KUKA KRL program: EPS_2_25369_MH1A_A_20251128065454.src

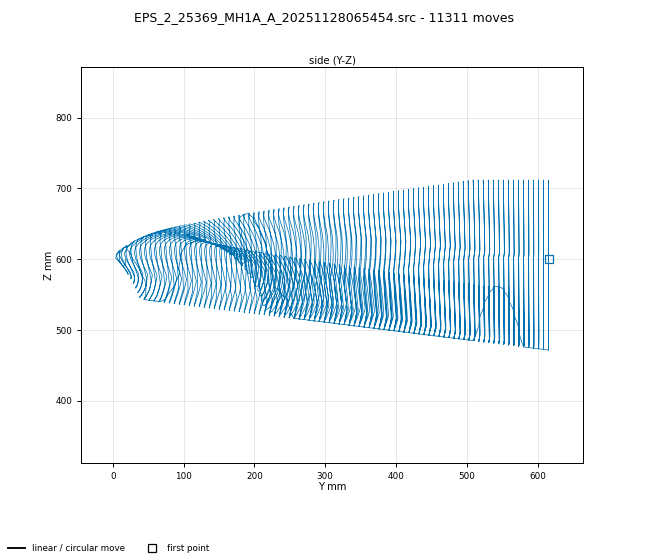
[picture p0: tool path of EPS_2_25369_MH1A_A_20251128065454.src, 11311 of 11313 moves have a stored position in this frame; points joined in program order, loops and branches not executed]
&ACCESS RVP
&REL 4
&COMMENT QRS 19112012
&PARAM EDITMASK = *
DEF PART()
EXT BAS (BAS_COMMAND :IN,REAL :IN )
INT I
BAS (#INITMOV,0 )

;KUKA QRS Post kuka4.cps  Date:22-06-2017 !

File_ID=2931

QRS_PRE_INIT()

;Init var - Until changes are made in qrs_pre_init
Outlet_Square_prg=0
Inlet_1_Square_prg=0
Inlet_2_Square_prg=0
Inlet_3_Square_prg=0
Inlet_4_Square_prg=0
Inlet_5_Square_prg=0

Outlet_1={X 0.000, Y 509.750, Z 611.500, B 0.000, E1 0.000 }
Inlet_1={X 0.000, Y 524.260, Z 411.500, B 0.000, E1 124.000 }
Outlet_1_type=201
Inlet_1_type=201
;QRS#1=Sidecore dimensions
;QRS#2=200-8" PVC SDR 35
;QRS#3=200-8" PVC SDR 35
;QRS#4=
;QRS#5=
;QRS#6=
;QRS#7=
;QRS#8=
;QRS#9=12-08 PSX
;QRS#10=12-08 PSX
;QRS#11=
;QRS#12=
;QRS#13=
;QRS#14=
;QRS#15=
;QRS#16=1220x127x991 3,25'
;QRS#17=EPS Height
;QRS#18=712
;QRS#19=*
;QRS#20= UPDATED VERSION 22-06-2017
;QRS#21=*
Outlet_Square=0100
Inlet_1_Square=0100
Inlet_2_Square=0
Inlet_3_Square=0
Inlet_4_Square=0
Inlet_5_Square=0
Mill_Square=1
Outlet_Square_Prg=204
Inlet_1_Square_prg=204

QRS_INIT()

$ADVANCE=5

; T1
PTP {E1 173.629,E2 173.629}
PTP {X 0,Y 615.476,A -85,B 0,C 180,E1 173.629,E2 173.629,E3 0,E4 0,E5 0,E6 0}
QRS_SPEED_INIT()
LIN {X 0,Y 615.476,Z 600,A -85,B 0,C 180,E1 173.629,E2 173.629,E3 0,E4 0,E5 0,E6 0} C_VEL
LIN {X 0,Y 615.476,Z 481.876,A -85,B 0,C 180,E1 173.629,E2 173.629} C_VEL
LIN {X 0,Y 615.476,Z 473.699,A -85,B 0,C 180,E1 173.629,E2 173.629} C_VEL
LIN {X 0,Y 615.467,Z 471.699,A -85,B 0,C 180,E1 173.442,E2 173.442} C_VEL
LIN {X 0,Y 615.466,Z 471.7,A -85,B 0,C 180,E1 170.801,E2 170.801} C_VEL
LIN {X 0,Y 615.488,Z 471.697,A -85,B 0,C 180,E1 168.139,E2 168.139} C_VEL
LIN {X 0,Y 615.489,Z 471.7,A -85,B 0,C 180,E1 165.451,E2 165.451} C_VEL
LIN {X 0,Y 615.49,Z 471.699,A -85,B 0,C 180,E1 162.729,E2 162.729} C_VEL
LIN {X 0,Y 615.492,Z 471.695,A -85,B 0,C 180,E1 159.967,E2 159.967} C_VEL
LIN {X 0,Y 615.461,Z 471.832,A -85,B 0,C 180,E1 157.233,E2 157.233} C_VEL
LIN {X 0,Y 615.482,Z 484.752,A -85,B 0,C 180,E1 156.799,E2 156.799} C_VEL
LIN {X 0,Y 615.487,Z 496.263,A -85,B 0,C 180,E1 156.274,E2 156.274} C_VEL
LIN {X 0,Y 615.488,Z 507.199,A -85,B 0,C 180,E1 155.638,E2 155.638} C_VEL
LIN {X 0,Y 615.498,Z 517.865,A -85,B 0,C 180,E1 154.864,E2 154.864} C_VEL
LIN {X 0,Y 615.497,Z 526.422,A -85,B 0,C 180,E1 154.103,E2 154.103} C_VEL
LIN {X 0,Y 615.499,Z 535.499,A -85,B 0,C 180,E1 153.105,E2 153.105} C_VEL
LIN {X 0,Y 615.497,Z 542.974,A -85,B 0,C 180,E1 152.085,E2 152.085} C_VEL
LIN {X 0,Y 615.497,Z 549.38,A -85,B 0,C 180,E1 150.969,E2 150.969} C_VEL
LIN {X 0,Y 615.495,Z 554.304,A -85,B 0,C 180,E1 149.84,E2 149.84} C_VEL
LIN {X 0,Y 615.493,Z 557.321,A -85,B 0,C 180,E1 148.914,E2 148.914} C_VEL
LIN {X 0,Y 615.496,Z 560.023,A -85,B 0,C 180,E1 147.669,E2 147.669} C_VEL
LIN {X 0,Y 615.494,Z 561.269,A -85,B 0,C 180,E1 146.466,E2 146.466} C_VEL
LIN {X 0,Y 615.497,Z 561.091,A -85,B 0,C 180,E1 145.185,E2 145.185} C_VEL
LIN {X 0,Y 615.496,Z 559.897,A -85,B 0,C 180,E1 144.166,E2 144.166} C_VEL
LIN {X 0,Y 615.495,Z 557.5,A -85,B 0,C 180,E1 143.063,E2 143.063} C_VEL
LIN {X 0,Y 615.497,Z 553.786,A -85,B 0,C 180,E1 141.932,E2 141.932} C_VEL
LIN {X 0,Y 615.497,Z 549.361,A -85,B 0,C 180,E1 140.937,E2 140.937} C_VEL
LIN {X 0,Y 615.497,Z 543.531,A -85,B 0,C 180,E1 139.91,E2 139.91} C_VEL
LIN {X 0,Y 615.495,Z 536.324,A -85,B 0,C 180,E1 138.905,E2 138.905} C_VEL
LIN {X 0,Y 615.498,Z 527.522,A -85,B 0,C 180,E1 137.919,E2 137.919} C_VEL
LIN {X 0,Y 615.499,Z 517.785,A -85,B 0,C 180,E1 137.04,E2 137.04} C_VEL
LIN {X 0,Y 615.492,Z 507.415,A -85,B 0,C 180,E1 136.286,E2 136.286} C_VEL
LIN {X 0,Y 615.48,Z 496.612,A -85,B 0,C 180,E1 135.654,E2 135.654} C_VEL
LIN {X 0,Y 615.493,Z 484.907,A -85,B 0,C 180,E1 135.117,E2 135.117} C_VEL
LIN {X 0,Y 615.477,Z 471.697,A -85,B 0,C 180,E1 134.663,E2 134.663} C_VEL
LIN {X 0,Y 615.488,Z 471.701,A -85,B 0,C 180,E1 132.08,E2 132.08} C_VEL
LIN {X 0,Y 615.483,Z 471.692,A -85,B 0,C 180,E1 129.751,E2 129.751} C_VEL
LIN {X 0,Y 615.466,Z 471.7,A -85,B 0,C 180,E1 127.244,E2 127.244} C_VEL
LIN {X 0,Y 615.483,Z 471.7,A -85,B 0,C 180,E1 124.699,E2 124.699} C_VEL
LIN {X 0,Y 615.476,Z 471.694,A -85,B 0,C 180,E1 122.328,E2 122.328} C_VEL
LIN {X 0,Y 615.454,Z 471.699,A -85,B 0,C 180,E1 119.408,E2 119.408} C_VEL
LIN {X 0,Y 615.497,Z 471.7,A -85,B 0,C 180,E1 117.046,E2 117.046} C_VEL
LIN {X 0,Y 615.474,Z 471.701,A -85,B 0,C 180,E1 114.273,E2 114.273} C_VEL
LIN {X 0,Y 615.482,Z 471.696,A -85,B 0,C 180,E1 111.432,E2 111.432} C_VEL
LIN {X 0,Y 615.47,Z 471.7,A -85,B 0,C 180,E1 109.339,E2 109.339} C_VEL
LIN {X 0,Y 615.491,Z 471.702,A -85,B 0,C 180,E1 106.587,E2 106.587} C_VEL
LIN {X 0,Y 615.495,Z 471.695,A -85,B 0,C 180,E1 103.874,E2 103.874} C_VEL
LIN {X 0,Y 615.474,Z 471.699,A -85,B 0,C 180,E1 100.878,E2 100.878} C_VEL
LIN {X 0,Y 615.47,Z 471.695,A -85,B 0,C 180,E1 98.537,E2 98.537} C_VEL
LIN {X 0,Y 615.487,Z 471.697,A -85,B 0,C 180,E1 95.899,E2 95.899} C_VEL
LIN {X 0,Y 615.491,Z 471.698,A -85,B 0,C 180,E1 93.273,E2 93.273} C_VEL
LIN {X 0,Y 615.452,Z 471.7,A -85,B 0,C 180,E1 90.654,E2 90.654} C_VEL
LIN {X 0,Y 615.498,Z 471.689,A -85,B 0,C 180,E1 88.037,E2 88.037} C_VEL
LIN {X 0,Y 615.471,Z 471.7,A -85,B 0,C 180,E1 85.415,E2 85.415} C_VEL
LIN {X 0,Y 615.482,Z 471.701,A -85,B 0,C 180,E1 82.784,E2 82.784} C_VEL
LIN {X 0,Y 615.486,Z 471.693,A -85,B 0,C 180,E1 80.138,E2 80.138} C_VEL
LIN {X 0,Y 615.461,Z 471.697,A -85,B 0,C 180,E1 77.469,E2 77.469} C_VEL
LIN {X 0,Y 615.487,Z 471.696,A -85,B 0,C 180,E1 75.451,E2 75.451} C_VEL
LIN {X 0,Y 615.453,Z 471.7,A -85,B 0,C 180,E1 72.728,E2 72.728} C_VEL
LIN {X 0,Y 615.491,Z 471.69,A -85,B 0,C 180,E1 69.967,E2 69.967} C_VEL
LIN {X 0,Y 615.451,Z 471.7,A -85,B 0,C 180,E1 67.154,E2 67.154} C_VEL
LIN {X 0,Y 615.486,Z 471.696,A -85,B 0,C 180,E1 64.433,E2 64.433} C_VEL
LIN {X 0,Y 615.478,Z 471.7,A -85,B 0,C 180,E1 61.552,E2 61.552} C_VEL
LIN {X 0,Y 615.482,Z 471.699,A -85,B 0,C 180,E1 58.916,E2 58.916} C_VEL
LIN {X 0,Y 615.464,Z 471.696,A -85,B 0,C 180,E1 56.47,E2 56.47} C_VEL
LIN {X 0,Y 615.468,Z 471.696,A -85,B 0,C 180,E1 53.574,E2 53.574} C_VEL
LIN {X 0,Y 615.472,Z 471.698,A -85,B 0,C 180,E1 50.94,E2 50.94} C_VEL
LIN {X 0,Y 615.471,Z 471.7,A -85,B 0,C 180,E1 48.525,E2 48.525} C_VEL
LIN {X 0,Y 615.492,Z 471.691,A -85,B 0,C 180,E1 45.851,E2 45.851} C_VEL
LIN {X 0,Y 615.448,Z 471.7,A -85,B 0,C 180,E1 43.043,E2 43.043} C_VEL
LIN {X 0,Y 615.485,Z 471.698,A -85,B 0,C 180,E1 40.607,E2 40.607} C_VEL
LIN {X 0,Y 615.486,Z 471.697,A -85,B 0,C 180,E1 38.012,E2 38.012} C_VEL
LIN {X 0,Y 615.471,Z 471.695,A -85,B 0,C 180,E1 35.617,E2 35.617} C_VEL
LIN {X 0,Y 615.485,Z 471.701,A -85,B 0,C 180,E1 33.237,E2 33.237} C_VEL
LIN {X 0,Y 615.449,Z 471.7,A -85,B 0,C 180,E1 30.922,E2 30.922} C_VEL
LIN {X 0,Y 615.484,Z 471.695,A -85,B 0,C 180,E1 28.449,E2 28.449} C_VEL
LIN {X 0,Y 615.47,Z 471.7,A -85,B 0,C 180,E1 25.565,E2 25.565} C_VEL
LIN {X 0,Y 615.487,Z 471.703,A -85,B 0,C 180,E1 22.845,E2 22.845} C_VEL
LIN {X 0,Y 615.487,Z 471.698,A -85,B 0,C 180,E1 20.033,E2 20.033} C_VEL
LIN {X 0,Y 615.472,Z 471.697,A -85,B 0,C 180,E1 17.271,E2 17.271} C_VEL
LIN {X 0,Y 615.482,Z 471.7,A -85,B 0,C 180,E1 15.226,E2 15.226} C_VEL
LIN {X 0,Y 615.477,Z 471.701,A -85,B 0,C 180,E1 12.531,E2 12.531} C_VEL
LIN {X 0,Y 615.493,Z 471.691,A -85,B 0,C 180,E1 9.862,E2 9.862} C_VEL
LIN {X 0,Y 615.449,Z 471.7,A -85,B 0,C 180,E1 7.216,E2 7.216} C_VEL
LIN {X 0,Y 615.484,Z 471.696,A -85,B 0,C 180,E1 4.585,E2 4.585} C_VEL
LIN {X 0,Y 615.499,Z 471.698,A -85,B 0,C 180,E1 1.963,E2 1.963} C_VEL
LIN {X 0,Y 615.473,Z 471.696,A -85,B 0,C 180,E1 -0.654,E2 -0.654} C_VEL
LIN {X 0,Y 615.452,Z 471.699,A -85,B 0,C 180,E1 -3.273,E2 -3.273} C_VEL
LIN {X 0,Y 615.496,Z 471.693,A -85,B 0,C 180,E1 -5.898,E2 -5.898} C_VEL
LIN {X 0,Y 615.491,Z 471.701,A -85,B 0,C 180,E1 -8.536,E2 -8.536} C_VEL
LIN {X 0,Y 615.461,Z 471.7,A -85,B 0,C 180,E1 -11.193,E2 -11.193} C_VEL
LIN {X 0,Y 615.495,Z 471.69,A -85,B 0,C 180,E1 -13.934,E2 -13.934} C_VEL
LIN {X 0,Y 615.45,Z 471.7,A -85,B 0,C 180,E1 -16.588,E2 -16.588} C_VEL
LIN {X 0,Y 615.476,Z 471.696,A -85,B 0,C 180,E1 -18.646,E2 -18.646} C_VEL
LIN {X 0,Y 615.475,Z 471.7,A -85,B 0,C 180,E1 -20.731,E2 -20.731} C_VEL
LIN {X 0,Y 615.485,Z 471.703,A -85,B 0,C 180,E1 -23.556,E2 -23.556} C_VEL
LIN {X 0,Y 615.478,Z 471.693,A -85,B 0,C 180,E1 -25.716,E2 -25.716} C_VEL
LIN {X 0,Y 615.449,Z 471.7,A -85,B 0,C 180,E1 -28.66,E2 -28.66} C_VEL
LIN {X 0,Y 615.484,Z 471.702,A -85,B 0,C 180,E1 -31.085,E2 -31.085} C_VEL
LIN {X 0,Y 615.455,Z 471.7,A -85,B 0,C 180,E1 -33.529,E2 -33.529} C_VEL
LIN {X 0,Y 615.475,Z 471.695,A -85,B 0,C 180,E1 -36.426,E2 -36.426} C_VEL
LIN {X 0,Y 615.451,Z 471.7,A -85,B 0,C 180,E1 -39.058,E2 -39.058} C_VEL
LIN {X 0,Y 615.494,Z 471.701,A -85,B 0,C 180,E1 -41.473,E2 -41.473} C_VEL
LIN {X 0,Y 615.494,Z 471.693,A -85,B 0,C 180,E1 -44.149,E2 -44.149} C_VEL
LIN {X 0,Y 615.454,Z 471.7,A -85,B 0,C 180,E1 -46.956,E2 -46.956} C_VEL
LIN {X 0,Y 615.476,Z 471.696,A -85,B 0,C 180,E1 -49.392,E2 -49.392} C_VEL
LIN {X 0,Y 615.48,Z 471.704,A -85,B 0,C 180,E1 -51.989,E2 -51.989} C_VEL
LIN {X 0,Y 615.479,Z 471.753,A -85,B 0,C 180,E1 -54.434,E2 -54.434} C_VEL
LIN {X 0,Y 615.486,Z 483.67,A -85,B 0,C 180,E1 -56.764,E2 -56.764} C_VEL
LIN {X 0,Y 615.477,Z 497.365,A -85,B 0,C 180,E1 -59.46,E2 -59.46} C_VEL
LIN {X 0,Y 615.49,Z 511.06,A -85,B 0,C 180,E1 -62.085,E2 -62.085} C_VEL
LIN {X 0,Y 615.449,Z 525.164,A -85,B 0,C 180,E1 -64.721,E2 -64.721} C_VEL
LIN {X 0,Y 615.486,Z 538.431,A -85,B 0,C 180,E1 -67.155,E2 -67.155} C_VEL
LIN {X 0,Y 615.469,Z 552.613,A -85,B 0,C 180,E1 -69.71,E2 -69.71} C_VEL
LIN {X 0,Y 615.477,Z 567.707,A -85,B 0,C 180,E1 -72.386,E2 -72.386} C_VEL
LIN {X 0,Y 615.47,Z 581.356,A -85,B 0,C 180,E1 -74.774,E2 -74.774} C_VEL
LIN {X 0,Y 615.487,Z 596.931,A -85,B 0,C 180,E1 -77.47,E2 -77.47} C_VEL
LIN {X 0,Y 615.481,Z 601.943,A -85,B 0,C 180,E1 -78.327,E2 -78.327} C_VEL
LIN {X 0,Y 615.479,Z 615.243,A -85,B 0,C 180,E1 -78.557,E2 -78.557} C_VEL
LIN {X 0,Y 615.497,Z 628.351,A -85,B 0,C 180,E1 -78.923,E2 -78.923} C_VEL
LIN {X 0,Y 615.473,Z 640.14,A -85,B 0,C 180,E1 -79.383,E2 -79.383} C_VEL
LIN {X 0,Y 615.489,Z 651.575,A -85,B 0,C 180,E1 -79.972,E2 -79.972} C_VEL
LIN {X 0,Y 615.499,Z 663.022,A -85,B 0,C 180,E1 -80.719,E2 -80.719} C_VEL
LIN {X 0,Y 615.498,Z 672.258,A -85,B 0,C 180,E1 -81.464,E2 -81.464} C_VEL
LIN {X 0,Y 615.499,Z 680.654,A -85,B 0,C 180,E1 -82.29,E2 -82.29} C_VEL
LIN {X 0,Y 615.497,Z 688.69,A -85,B 0,C 180,E1 -83.259,E2 -83.259} C_VEL
LIN {X 0,Y 615.498,Z 694.423,A -85,B 0,C 180,E1 -84.102,E2 -84.102} C_VEL
LIN {X 0,Y 615.496,Z 699.873,A -85,B 0,C 180,E1 -85.087,E2 -85.087} C_VEL
LIN {X 0,Y 615.497,Z 704.141,A -85,B 0,C 180,E1 -86.072,E2 -86.072} C_VEL
LIN {X 0,Y 615.494,Z 706.399,A -85,B 0,C 180,E1 -86.727,E2 -86.727} C_VEL
LIN {X 0,Y 615.497,Z 708.233,A -85,B 0,C 180,E1 -87.382,E2 -87.382} C_VEL
LIN {X 0,Y 615.499,Z 709.608,A -85,B 0,C 180,E1 -88.037,E2 -88.037} C_VEL
LIN {X 0,Y 615.496,Z 711.174,A -85,B 0,C 180,E1 -89.346,E2 -89.346} C_VEL
LIN {X 0,Y 615.494,Z 711.389,A -85,B 0,C 180,E1 -90,E2 -90} C_VEL
LIN {X 0,Y 615.495,Z 710.58,A -85,B 0,C 180,E1 -91.309,E2 -91.309} C_VEL
LIN {X 0,Y 615.499,Z 709.608,A -85,B 0,C 180,E1 -91.963,E2 -91.963} C_VEL
LIN {X 0,Y 615.497,Z 708.233,A -85,B 0,C 180,E1 -92.618,E2 -92.618} C_VEL
LIN {X 0,Y 615.496,Z 705.349,A -85,B 0,C 180,E1 -93.601,E2 -93.601} C_VEL
LIN {X 0,Y 615.498,Z 701.441,A -85,B 0,C 180,E1 -94.585,E2 -94.585} C_VEL
LIN {X 0,Y 615.499,Z 696.404,A -85,B 0,C 180,E1 -95.57,E2 -95.57} C_VEL
LIN {X 0,Y 615.497,Z 689.869,A -85,B 0,C 180,E1 -96.583,E2 -96.583} C_VEL
LIN {X 0,Y 615.497,Z 682.132,A -85,B 0,C 180,E1 -97.546,E2 -97.546} C_VEL
LIN {X 0,Y 615.498,Z 674.043,A -85,B 0,C 180,E1 -98.371,E2 -98.371} C_VEL
LIN {X 0,Y 615.499,Z 664.165,A -85,B 0,C 180,E1 -99.199,E2 -99.199} C_VEL
LIN {X 0,Y 615.491,Z 652.978,A -85,B 0,C 180,E1 -99.945,E2 -99.945} C_VEL
LIN {X 0,Y 615.473,Z 642.022,A -85,B 0,C 180,E1 -100.527,E2 -100.527} C_VEL
LIN {X 0,Y 615.495,Z 629.52,A -85,B 0,C 180,E1 -101.039,E2 -101.039} C_VEL
LIN {X 0,Y 615.48,Z 617.06,A -85,B 0,C 180,E1 -101.402,E2 -101.402} C_VEL
LIN {X 0,Y 615.48,Z 603.456,A -85,B 0,C 180,E1 -101.652,E2 -101.652} C_VEL
LIN {X 0,Y 615.481,Z 601.797,A -85,B 0,C 180,E1 -101.694,E2 -101.694} C_VEL
LIN {X 0,Y 615.453,Z 585.25,A -85,B 0,C 180,E1 -104.55,E2 -104.55} C_VEL
LIN {X 0,Y 615.496,Z 571.604,A -85,B 0,C 180,E1 -106.928,E2 -106.928} C_VEL
LIN {X 0,Y 615.47,Z 556.004,A -85,B 0,C 180,E1 -109.686,E2 -109.686} C_VEL
LIN {X 0,Y 615.482,Z 541.192,A -85,B 0,C 180,E1 -112.344,E2 -112.344} C_VEL
LIN {X 0,Y 615.449,Z 526.706,A -85,B 0,C 180,E1 -114.994,E2 -114.994} C_VEL
LIN {X 0,Y 615.493,Z 513.016,A -85,B 0,C 180,E1 -117.545,E2 -117.545} C_VEL
LIN {X 0,Y 615.492,Z 499.321,A -85,B 0,C 180,E1 -120.16,E2 -120.16} C_VEL
LIN {X 0,Y 615.46,Z 485.626,A -85,B 0,C 180,E1 -122.848,E2 -122.848} C_VEL
LIN {X 0,Y 615.493,Z 475.538,A -85,B 0,C 180,E1 -124.815,E2 -124.815} C_VEL
LIN {X 0,Y 615.477,Z 471.697,A -85,B 0,C 180,E1 -125.567,E2 -125.567} C_VEL
LIN {X 0,Y 615.49,Z 471.694,A -85,B 0,C 180,E1 -128.069,E2 -128.069} C_VEL
LIN {X 0,Y 615.466,Z 471.7,A -85,B 0,C 180,E1 -130.609,E2 -130.609} C_VEL
LIN {X 0,Y 615.467,Z 471.7,A -85,B 0,C 180,E1 -133.247,E2 -133.247} C_VEL
LIN {X 0,Y 615.49,Z 471.698,A -85,B 0,C 180,E1 -136.003,E2 -136.003} C_VEL
LIN {X 0,Y 615.491,Z 471.699,A -85,B 0,C 180,E1 -138.526,E2 -138.526} C_VEL
LIN {X 0,Y 615.488,Z 471.701,A -85,B 0,C 180,E1 -141.096,E2 -141.096} C_VEL
LIN {X 0,Y 615.486,Z 471.701,A -85,B 0,C 180,E1 -143.575,E2 -143.575} C_VEL
LIN {X 0,Y 615.472,Z 471.7,A -85,B 0,C 180,E1 -146.469,E2 -146.469} C_VEL
LIN {X 0,Y 615.467,Z 471.7,A -85,B 0,C 180,E1 -149.079,E2 -149.079} C_VEL
LIN {X 0,Y 615.482,Z 471.697,A -85,B 0,C 180,E1 -151.552,E2 -151.552} C_VEL
LIN {X 0,Y 615.482,Z 471.697,A -85,B 0,C 180,E1 -154.433,E2 -154.433} C_VEL
LIN {X 0,Y 615.482,Z 471.7,A -85,B 0,C 180,E1 -157.155,E2 -157.155} C_VEL
LIN {X 0,Y 615.492,Z 471.698,A -85,B 0,C 180,E1 -159.967,E2 -159.967} C_VEL
LIN {X 0,Y 615.468,Z 471.7,A -85,B 0,C 180,E1 -162.729,E2 -162.729} C_VEL
LIN {X 0,Y 615.467,Z 471.699,A -85,B 0,C 180,E1 -165.451,E2 -165.451} C_VEL
LIN {X 0,Y 615.495,Z 471.694,A -85,B 0,C 180,E1 -168.139,E2 -168.139} C_VEL
LIN {X 0,Y 615.478,Z 471.7,A -85,B 0,C 180,E1 -170.801,E2 -170.801} C_VEL
LIN {X 0,Y 615.493,Z 471.7,A -85,B 0,C 180,E1 -173.444,E2 -173.444} C_VEL
LIN {X 0,Y 615.484,Z 471.702,A -85,B 0,C 180,E1 -176.072,E2 -176.072} C_VEL
LIN {X 0,Y 615.48,Z 471.7,A -85,B 0,C 180,E1 -178.692,E2 -178.692} C_VEL
LIN {X 0,Y 615.479,Z 471.698,A -85,B 0,C 180,E1 -181.309,E2 -181.309} C_VEL
LIN {X 0,Y 615.491,Z 471.695,A -85,B 0,C 180,E1 -183.929,E2 -183.929} C_VEL
LIN {X 0,Y 615.467,Z 471.699,A -85,B 0,C 180,E1 -186.558,E2 -186.558} C_VEL
LIN {X 0,Y 614.8,Z 471.848,A -85,B 0,C 180,E1 -187.104,E2 -187.104} C_VEL
LIN {X 0,Y 611.963,Z 472.257,A -85,B 0,C 180,E1 -187.99,E2 -187.99} C_VEL
LIN {X 0,Y 609.567,Z 472.567,A -85,B 0,C 180,E1 -188.702,E2 -188.702} C_VEL
LIN {X 0,Y 608.536,Z 472.685,A -85,B 0,C 180,E1 -189.252,E2 -189.252} C_VEL
LIN {X 0,Y 608.451,Z 472.694,A -85,B 0,C 180,E1 -189.438,E2 -189.438} C_VEL
LIN {X 0,Y 608.461,Z 472.695,A -85,B 0,C 180,E1 -192,E2 -192} C_VEL
LIN {X 0,Y 608.473,Z 472.695,A -85,B 0,C 180,E1 -194.721,E2 -194.721} C_VEL
LIN {X 0,Y 608.458,Z 472.694,A -85,B 0,C 180,E1 -197.477,E2 -197.477} C_VEL
LIN {X 0,Y 608.464,Z 472.693,A -85,B 0,C 180,E1 -200.274,E2 -200.274} C_VEL
LIN {X 0,Y 608.433,Z 472.697,A -85,B 0,C 180,E1 -202.642,E2 -202.642} C_VEL
LIN {X 0,Y 608.52,Z 487.034,A -85,B 0,C 180,E1 -203.167,E2 -203.167} C_VEL
LIN {X 0,Y 608.502,Z 499.16,A -85,B 0,C 180,E1 -203.753,E2 -203.753} C_VEL
LIN {X 0,Y 608.475,Z 510.181,A -85,B 0,C 180,E1 -204.434,E2 -204.434} C_VEL
LIN {X 0,Y 608.466,Z 521.281,A -85,B 0,C 180,E1 -205.301,E2 -205.301} C_VEL
LIN {X 0,Y 608.469,Z 530.757,A -85,B 0,C 180,E1 -206.219,E2 -206.219} C_VEL
LIN {X 0,Y 608.441,Z 538.894,A -85,B 0,C 180,E1 -207.199,E2 -207.199} C_VEL
LIN {X 0,Y 608.447,Z 546.017,A -85,B 0,C 180,E1 -208.267,E2 -208.267} C_VEL
LIN {X 0,Y 608.432,Z 551.923,A -85,B 0,C 180,E1 -209.401,E2 -209.401} C_VEL
LIN {X 0,Y 608.433,Z 556.359,A -85,B 0,C 180,E1 -210.547,E2 -210.547} C_VEL
LIN {X 0,Y 608.424,Z 558.605,A -85,B 0,C 180,E1 -211.319,E2 -211.319} C_VEL
LIN {X 0,Y 608.419,Z 560.94,A -85,B 0,C 180,E1 -212.515,E2 -212.515} C_VEL
LIN {X 0,Y 608.418,Z 561.931,A -85,B 0,C 180,E1 -213.727,E2 -213.727} C_VEL
LIN {X 0,Y 608.421,Z 561.647,A -85,B 0,C 180,E1 -214.901,E2 -214.901} C_VEL
LIN {X 0,Y 608.424,Z 560.096,A -85,B 0,C 180,E1 -216.094,E2 -216.094} C_VEL
LIN {X 0,Y 608.435,Z 557.581,A -85,B 0,C 180,E1 -217.153,E2 -217.153} C_VEL
LIN {X 0,Y 608.43,Z 553.86,A -85,B 0,C 180,E1 -218.235,E2 -218.235} C_VEL
LIN {X 0,Y 608.458,Z 548.164,A -85,B 0,C 180,E1 -219.441,E2 -219.441} C_VEL
LIN {X 0,Y 608.447,Z 541.551,A -85,B 0,C 180,E1 -220.521,E2 -220.521} C_VEL
LIN {X 0,Y 608.452,Z 534.226,A -85,B 0,C 180,E1 -221.48,E2 -221.48} C_VEL
LIN {X 0,Y 608.476,Z 525.045,A -85,B 0,C 180,E1 -222.447,E2 -222.447} C_VEL
LIN {X 0,Y 608.497,Z 514.91,A -85,B 0,C 180,E1 -223.311,E2 -223.311} C_VEL
LIN {X 0,Y 608.495,Z 503.803,A -85,B 0,C 180,E1 -224.068,E2 -224.068} C_VEL
LIN {X 0,Y 608.494,Z 491.815,A -85,B 0,C 180,E1 -224.712,E2 -224.712} C_VEL
LIN {X 0,Y 608.534,Z 479.655,A -85,B 0,C 180,E1 -225.211,E2 -225.211} C_VEL
LIN {X 0,Y 608.472,Z 472.691,A -85,B 0,C 180,E1 -225.446,E2 -225.446} C_VEL
LIN {X 0,Y 608.467,Z 472.696,A -85,B 0,C 180,E1 -227.939,E2 -227.939} C_VEL
LIN {X 0,Y 608.451,Z 472.695,A -85,B 0,C 180,E1 -230.705,E2 -230.705} C_VEL
LIN {X 0,Y 608.42,Z 472.696,A -85,B 0,C 180,E1 -233.082,E2 -233.082} C_VEL
LIN {X 0,Y 608.471,Z 472.695,A -85,B 0,C 180,E1 -235.531,E2 -235.531} C_VEL
LIN {X 0,Y 608.464,Z 472.691,A -85,B 0,C 180,E1 -237.905,E2 -237.905} C_VEL
LIN {X 0,Y 608.462,Z 472.693,A -85,B 0,C 180,E1 -240.22,E2 -240.22} C_VEL
LIN {X 0,Y 608.486,Z 472.692,A -85,B 0,C 180,E1 -242.793,E2 -242.793} C_VEL
LIN {X 0,Y 608.435,Z 472.695,A -85,B 0,C 180,E1 -245.428,E2 -245.428} C_VEL
LIN {X 0,Y 608.47,Z 472.69,A -85,B 0,C 180,E1 -248.308,E2 -248.308} C_VEL
LIN {X 0,Y 608.441,Z 472.693,A -85,B 0,C 180,E1 -251.13,E2 -251.13} C_VEL
LIN {X 0,Y 608.463,Z 472.691,A -85,B 0,C 180,E1 -253.906,E2 -253.906} C_VEL
LIN {X 0,Y 608.446,Z 472.696,A -85,B 0,C 180,E1 -256.643,E2 -256.643} C_VEL
LIN {X 0,Y 608.463,Z 472.697,A -85,B 0,C 180,E1 -259.35,E2 -259.35} C_VEL
LIN {X 0,Y 608.484,Z 472.69,A -85,B 0,C 180,E1 -262.033,E2 -262.033} C_VEL
LIN {X 0,Y 608.442,Z 472.693,A -85,B 0,C 180,E1 -264.698,E2 -264.698} C_VEL
LIN {X 0,Y 608.462,Z 472.692,A -85,B 0,C 180,E1 -267.352,E2 -267.352} C_VEL
LIN {X 0,Y 608.481,Z 472.693,A -85,B 0,C 180,E1 -270,E2 -270} C_VEL
LIN {X 0,Y 608.476,Z 472.693,A -85,B 0,C 180,E1 -272.648,E2 -272.648} C_VEL
LIN {X 0,Y 608.437,Z 472.695,A -85,B 0,C 180,E1 -275.302,E2 -275.302} C_VEL
LIN {X 0,Y 608.483,Z 472.688,A -85,B 0,C 180,E1 -277.967,E2 -277.967} C_VEL
LIN {X 0,Y 608.446,Z 472.695,A -85,B 0,C 180,E1 -280.65,E2 -280.65} C_VEL
LIN {X 0,Y 608.467,Z 472.696,A -85,B 0,C 180,E1 -283.356,E2 -283.356} C_VEL
LIN {X 0,Y 608.461,Z 472.694,A -85,B 0,C 180,E1 -286.094,E2 -286.094} C_VEL
LIN {X 0,Y 608.449,Z 472.694,A -85,B 0,C 180,E1 -288.87,E2 -288.87} C_VEL
LIN {X 0,Y 608.461,Z 472.691,A -85,B 0,C 180,E1 -291.692,E2 -291.692} C_VEL
LIN {X 0,Y 608.445,Z 472.693,A -85,B 0,C 180,E1 -294.571,E2 -294.571} C_VEL
LIN {X 0,Y 608.447,Z 472.694,A -85,B 0,C 180,E1 -297.2,E2 -297.2} C_VEL
LIN {X 0,Y 608.474,Z 472.693,A -85,B 0,C 180,E1 -299.971,E2 -299.971} C_VEL
LIN {X 0,Y 608.45,Z 472.697,A -85,B 0,C 180,E1 -302.88,E2 -302.88} C_VEL
LIN {X 0,Y 608.43,Z 472.696,A -85,B 0,C 180,E1 -305.279,E2 -305.279} C_VEL
LIN {X 0,Y 608.473,Z 472.69,A -85,B 0,C 180,E1 -307.746,E2 -307.746} C_VEL
LIN {X 0,Y 608.447,Z 472.698,A -85,B 0,C 180,E1 -310.328,E2 -310.328} C_VEL
LIN {X 0,Y 608.486,Z 472.693,A -85,B 0,C 180,E1 -313.31,E2 -313.31} C_VEL
LIN {X 0,Y 608.47,Z 472.695,A -85,B 0,C 180,E1 -316.13,E2 -316.13} C_VEL
LIN {X 0,Y 608.442,Z 472.695,A -85,B 0,C 180,E1 -318.822,E2 -318.822} C_VEL
LIN {X 0,Y 608.464,Z 472.692,A -85,B 0,C 180,E1 -321.76,E2 -321.76} C_VEL
LIN {X 0,Y 608.44,Z 472.694,A -85,B 0,C 180,E1 -324.722,E2 -324.722} C_VEL
LIN {X 0,Y 608.45,Z 472.694,A -85,B 0,C 180,E1 -327.12,E2 -327.12} C_VEL
LIN {X 0,Y 608.469,Z 472.692,A -85,B 0,C 180,E1 -330.029,E2 -330.029} C_VEL
LIN {X 0,Y 608.474,Z 472.694,A -85,B 0,C 180,E1 -332.794,E2 -332.794} C_VEL
LIN {X 0,Y 608.443,Z 472.696,A -85,B 0,C 180,E1 -335.428,E2 -335.428} C_VEL
LIN {X 0,Y 608.475,Z 472.691,A -85,B 0,C 180,E1 -338.308,E2 -338.308} C_VEL
LIN {X 0,Y 608.442,Z 472.695,A -85,B 0,C 180,E1 -341.293,E2 -341.293} C_VEL
LIN {X 0,Y 608.463,Z 472.691,A -85,B 0,C 180,E1 -343.906,E2 -343.906} C_VEL
LIN {X 0,Y 608.44,Z 472.694,A -85,B 0,C 180,E1 -346.643,E2 -346.643} C_VEL
LIN {X 0,Y 608.463,Z 472.694,A -85,B 0,C 180,E1 -349.35,E2 -349.35} C_VEL
LIN {X 0,Y 608.476,Z 472.694,A -85,B 0,C 180,E1 -352.033,E2 -352.033} C_VEL
LIN {X 0,Y 608.457,Z 472.693,A -85,B 0,C 180,E1 -354.698,E2 -354.698} C_VEL
LIN {X 0,Y 608.448,Z 472.693,A -85,B 0,C 180,E1 -357.352,E2 -357.352} C_VEL
LIN {X 0,Y 608.48,Z 472.69,A -85,B 0,C 180,E1 -360,E2 -360} C_VEL
LIN {X 0,Y 608.481,Z 472.694,A -85,B 0,C 180,E1 -362.648,E2 -362.648} C_VEL
LIN {X 0,Y 608.446,Z 472.695,A -85,B 0,C 180,E1 -365.302,E2 -365.302} C_VEL
LIN {X 0,Y 608.481,Z 472.689,A -85,B 0,C 180,E1 -367.967,E2 -367.967} C_VEL
LIN {X 0,Y 608.444,Z 472.693,A -85,B 0,C 180,E1 -370.942,E2 -370.942} C_VEL
LIN {X 0,Y 608.466,Z 472.693,A -85,B 0,C 180,E1 -373.356,E2 -373.356} C_VEL
LIN {X 0,Y 608.45,Z 472.698,A -85,B 0,C 180,E1 -376.094,E2 -376.094} C_VEL
LIN {X 0,Y 608.452,Z 472.696,A -85,B 0,C 180,E1 -378.87,E2 -378.87} C_VEL
LIN {X 0,Y 608.451,Z 472.694,A -85,B 0,C 180,E1 -381.692,E2 -381.692} C_VEL
LIN {X 0,Y 608.453,Z 472.693,A -85,B 0,C 180,E1 -384.571,E2 -384.571} C_VEL
LIN {X 0,Y 608.431,Z 472.695,A -85,B 0,C 180,E1 -387.198,E2 -387.198} C_VEL
LIN {X 0,Y 608.473,Z 472.69,A -85,B 0,C 180,E1 -389.972,E2 -389.972} C_VEL
LIN {X 0,Y 608.442,Z 472.695,A -85,B 0,C 180,E1 -392.88,E2 -392.88} C_VEL
LIN {X 0,Y 608.435,Z 472.697,A -85,B 0,C 180,E1 -395.278,E2 -395.278} C_VEL
LIN {X 0,Y 608.471,Z 472.69,A -85,B 0,C 180,E1 -397.746,E2 -397.746} C_VEL
LIN {X 0,Y 608.435,Z 472.696,A -85,B 0,C 180,E1 -400.327,E2 -400.327} C_VEL
LIN {X 0,Y 608.453,Z 472.698,A -85,B 0,C 180,E1 -402.96,E2 -402.96} C_VEL
LIN {X 0,Y 608.451,Z 472.695,A -85,B 0,C 180,E1 -405.737,E2 -405.737} C_VEL
LIN {X 0,Y 608.459,Z 472.693,A -85,B 0,C 180,E1 -408.658,E2 -408.658} C_VEL
LIN {X 0,Y 608.461,Z 472.695,A -85,B 0,C 180,E1 -411.761,E2 -411.761} C_VEL
LIN {X 0,Y 608.496,Z 472.788,A -85,B 0,C 180,E1 -414.251,E2 -414.251} C_VEL
LIN {X 0,Y 608.628,Z 484.561,A -85,B 0,C 180,E1 -416.538,E2 -416.538} C_VEL
LIN {X 0,Y 608.591,Z 495.51,A -85,B 0,C 180,E1 -418.71,E2 -418.71} C_VEL
LIN {X 0,Y 608.591,Z 509.083,A -85,B 0,C 180,E1 -421.36,E2 -421.36} C_VEL
LIN {X 0,Y 608.553,Z 524.365,A -85,B 0,C 180,E1 -424.264,E2 -424.264} C_VEL
LIN {X 0,Y 608.533,Z 538.45,A -85,B 0,C 180,E1 -426.879,E2 -426.879} C_VEL
LIN {X 0,Y 608.471,Z 552.985,A -85,B 0,C 180,E1 -429.525,E2 -429.525} C_VEL
LIN {X 0,Y 608.478,Z 567.797,A -85,B 0,C 180,E1 -432.177,E2 -432.177} C_VEL
LIN {X 0,Y 608.445,Z 583.448,A -85,B 0,C 180,E1 -434.936,E2 -434.936} C_VEL
LIN {X 0,Y 608.453,Z 599.1,A -85,B 0,C 180,E1 -437.662,E2 -437.662} C_VEL
LIN {X 0,Y 608.448,Z 602.157,A -85,B 0,C 180,E1 -438.19,E2 -438.19} C_VEL
LIN {X 0,Y 608.526,Z 615.354,A -85,B 0,C 180,E1 -438.424,E2 -438.424} C_VEL
LIN {X 0,Y 608.532,Z 627.936,A -85,B 0,C 180,E1 -438.777,E2 -438.777} C_VEL
LIN {X 0,Y 608.508,Z 639.046,A -85,B 0,C 180,E1 -439.207,E2 -439.207} C_VEL
LIN {X 0,Y 608.502,Z 650.328,A -85,B 0,C 180,E1 -439.771,E2 -439.771} C_VEL
LIN {X 0,Y 608.491,Z 660.93,A -85,B 0,C 180,E1 -440.443,E2 -440.443} C_VEL
LIN {X 0,Y 608.477,Z 670.599,A -85,B 0,C 180,E1 -441.197,E2 -441.197} C_VEL
LIN {X 0,Y 608.46,Z 679.414,A -85,B 0,C 180,E1 -442.033,E2 -442.033} C_VEL
LIN {X 0,Y 608.444,Z 687.998,A -85,B 0,C 180,E1 -443.034,E2 -443.034} C_VEL
LIN {X 0,Y 608.438,Z 694.866,A -85,B 0,C 180,E1 -444.033,E2 -444.033} C_VEL
LIN {X 0,Y 608.437,Z 700.365,A -85,B 0,C 180,E1 -445.03,E2 -445.03} C_VEL
LIN {X 0,Y 608.435,Z 704.676,A -85,B 0,C 180,E1 -446.026,E2 -446.026} C_VEL
LIN {X 0,Y 608.424,Z 706.956,A -85,B 0,C 180,E1 -446.689,E2 -446.689} C_VEL
LIN {X 0,Y 608.425,Z 708.809,A -85,B 0,C 180,E1 -447.352,E2 -447.352} C_VEL
LIN {X 0,Y 608.444,Z 710.201,A -85,B 0,C 180,E1 -448.014,E2 -448.014} C_VEL
LIN {X 0,Y 608.438,Z 711.784,A -85,B 0,C 180,E1 -449.338,E2 -449.338} C_VEL
LIN {X 0,Y 608.434,Z 712,A -85,B 0,C 180,E1 -450,E2 -450} C_VEL
LIN {X 0,Y 608.448,Z 711.184,A -85,B 0,C 180,E1 -451.324,E2 -451.324} C_VEL
LIN {X 0,Y 608.444,Z 710.201,A -85,B 0,C 180,E1 -451.986,E2 -451.986} C_VEL
LIN {X 0,Y 608.425,Z 708.809,A -85,B 0,C 180,E1 -452.648,E2 -452.648} C_VEL
LIN {X 0,Y 608.449,Z 705.896,A -85,B 0,C 180,E1 -453.642,E2 -453.642} C_VEL
LIN {X 0,Y 608.432,Z 701.95,A -85,B 0,C 180,E1 -454.638,E2 -454.638} C_VEL
LIN {X 0,Y 608.437,Z 695.876,A -85,B 0,C 180,E1 -455.801,E2 -455.801} C_VEL
LIN {X 0,Y 608.462,Z 689.234,A -85,B 0,C 180,E1 -456.799,E2 -456.799} C_VEL
LIN {X 0,Y 608.456,Z 680.988,A -85,B 0,C 180,E1 -457.8,E2 -457.8} C_VEL
LIN {X 0,Y 608.472,Z 672.534,A -85,B 0,C 180,E1 -458.636,E2 -458.636} C_VEL
LIN {X 0,Y 608.481,Z 662.089,A -85,B 0,C 180,E1 -459.473,E2 -459.473} C_VEL
LIN {X 0,Y 608.496,Z 651.753,A -85,B 0,C 180,E1 -460.145,E2 -460.145} C_VEL
LIN {X 0,Y 608.501,Z 640.278,A -85,B 0,C 180,E1 -460.74,E2 -460.74} C_VEL
LIN {X 0,Y 608.532,Z 627.931,A -85,B 0,C 180,E1 -461.223,E2 -461.223} C_VEL
LIN {X 0,Y 608.537,Z 614.432,A -85,B 0,C 180,E1 -461.597,E2 -461.597} C_VEL
LIN {X 0,Y 608.448,Z 602.156,A -85,B 0,C 180,E1 -461.81,E2 -461.81} C_VEL
LIN {X 0,Y 608.448,Z 587.36,A -85,B 0,C 180,E1 -464.379,E2 -464.379} C_VEL
LIN {X 0,Y 608.476,Z 571.709,A -85,B 0,C 180,E1 -467.13,E2 -467.13} C_VEL
LIN {X 0,Y 608.481,Z 556.057,A -85,B 0,C 180,E1 -469.921,E2 -469.921} C_VEL
LIN {X 0,Y 608.525,Z 540.408,A -85,B 0,C 180,E1 -472.762,E2 -472.762} C_VEL
LIN {X 0,Y 608.528,Z 526.711,A -85,B 0,C 180,E1 -475.298,E2 -475.298} C_VEL
LIN {X 0,Y 608.604,Z 511.059,A -85,B 0,C 180,E1 -478.259,E2 -478.259} C_VEL
LIN {X 0,Y 608.58,Z 497.415,A -85,B 0,C 180,E1 -480.914,E2 -480.914} C_VEL
LIN {X 0,Y 608.651,Z 485.61,A -85,B 0,C 180,E1 -483.263,E2 -483.263} C_VEL
LIN {X 0,Y 608.474,Z 472.693,A -85,B 0,C 180,E1 -485.682,E2 -485.682} C_VEL
LIN {X 0,Y 608.467,Z 472.695,A -85,B 0,C 180,E1 -488.589,E2 -488.589} C_VEL
LIN {X 0,Y 608.46,Z 472.696,A -85,B 0,C 180,E1 -491.342,E2 -491.342} C_VEL
LIN {X 0,Y 608.459,Z 472.693,A -85,B 0,C 180,E1 -494.264,E2 -494.264} C_VEL
LIN {X 0,Y 608.434,Z 472.697,A -85,B 0,C 180,E1 -497.038,E2 -497.038} C_VEL
LIN {X 0,Y 608.456,Z 472.695,A -85,B 0,C 180,E1 -499.697,E2 -499.697} C_VEL
LIN {X 0,Y 608.467,Z 472.695,A -85,B 0,C 180,E1 -502.254,E2 -502.254} C_VEL
LIN {X 0,Y 608.443,Z 472.697,A -85,B 0,C 180,E1 -505.096,E2 -505.096} C_VEL
LIN {X 0,Y 608.471,Z 472.692,A -85,B 0,C 180,E1 -507.906,E2 -507.906} C_VEL
LIN {X 0,Y 608.468,Z 472.693,A -85,B 0,C 180,E1 -510.22,E2 -510.22} C_VEL
LIN {X 0,Y 608.464,Z 472.693,A -85,B 0,C 180,E1 -512.796,E2 -512.796} C_VEL
LIN {X 0,Y 608.45,Z 472.694,A -85,B 0,C 180,E1 -515.429,E2 -515.429} C_VEL
LIN {X 0,Y 608.478,Z 472.692,A -85,B 0,C 180,E1 -518.309,E2 -518.309} C_VEL
LIN {X 0,Y 608.471,Z 472.694,A -85,B 0,C 180,E1 -521.285,E2 -521.285} C_VEL
LIN {X 0,Y 608.466,Z 472.693,A -85,B 0,C 180,E1 -523.906,E2 -523.906} C_VEL
LIN {X 0,Y 608.451,Z 472.694,A -85,B 0,C 180,E1 -526.643,E2 -526.643} C_VEL
LIN {X 0,Y 608.45,Z 472.695,A -85,B 0,C 180,E1 -529.35,E2 -529.35} C_VEL
LIN {X 0,Y 608.485,Z 472.692,A -85,B 0,C 180,E1 -532.033,E2 -532.033} C_VEL
LIN {X 0,Y 608.473,Z 472.695,A -85,B 0,C 180,E1 -534.698,E2 -534.698} C_VEL
LIN {X 0,Y 608.479,Z 472.694,A -85,B 0,C 180,E1 -537.352,E2 -537.352} C_VEL
LIN {X 0,Y 608.482,Z 472.692,A -85,B 0,C 180,E1 -540,E2 -540} C_VEL
LIN {X 0,Y 608.462,Z 472.693,A -85,B 0,C 180,E1 -542.648,E2 -542.648} C_VEL
LIN {X 0,Y 608.446,Z 472.695,A -85,B 0,C 180,E1 -545.302,E2 -545.302} C_VEL
LIN {X 0,Y 608.482,Z 472.691,A -85,B 0,C 180,E1 -547.967,E2 -547.967} C_VEL
LIN {X 0,Y 608.451,Z 472.694,A -85,B 0,C 180,E1 -549.438,E2 -549.438} C_VEL
LIN {X 0,Y 607.783,Z 472.779,A -85,B 0,C 180,E1 -549.991,E2 -549.991} C_VEL
LIN {X 0,Y 604.936,Z 473.136,A -85,B 0,C 180,E1 -550.888,E2 -550.888} C_VEL
LIN {X 0,Y 602.529,Z 473.437,A -85,B 0,C 180,E1 -551.609,E2 -551.609} C_VEL
LIN {X 0,Y 601.492,Z 473.565,A -85,B 0,C 180,E1 -552.166,E2 -552.166} C_VEL
LIN {X 0,Y 601.405,Z 473.573,A -85,B 0,C 180,E1 -552.354,E2 -552.354} C_VEL
LIN {X 0,Y 601.426,Z 473.571,A -85,B 0,C 180,E1 -554.897,E2 -554.897} C_VEL
LIN {X 0,Y 601.402,Z 473.573,A -85,B 0,C 180,E1 -557.688,E2 -557.688} C_VEL
LIN {X 0,Y 601.433,Z 473.57,A -85,B 0,C 180,E1 -560.522,E2 -560.522} C_VEL
LIN {X 0,Y 601.425,Z 473.573,A -85,B 0,C 180,E1 -562.546,E2 -562.546} C_VEL
LIN {X 0,Y 601.547,Z 486.024,A -85,B 0,C 180,E1 -562.996,E2 -562.996} C_VEL
LIN {X 0,Y 601.51,Z 496.682,A -85,B 0,C 180,E1 -563.498,E2 -563.498} C_VEL
LIN {X 0,Y 601.468,Z 507.488,A -85,B 0,C 180,E1 -564.14,E2 -564.14} C_VEL
LIN {X 0,Y 601.44,Z 518.658,A -85,B 0,C 180,E1 -564.97,E2 -564.97} C_VEL
LIN {X 0,Y 601.404,Z 528.879,A -85,B 0,C 180,E1 -565.928,E2 -565.928} C_VEL
LIN {X 0,Y 601.387,Z 537.464,A -85,B 0,C 180,E1 -566.927,E2 -566.927} C_VEL
LIN {X 0,Y 601.357,Z 544.044,A -85,B 0,C 180,E1 -567.871,E2 -567.871} C_VEL
LIN {X 0,Y 601.337,Z 550.576,A -85,B 0,C 180,E1 -569.06,E2 -569.06} C_VEL
LIN {X 0,Y 601.354,Z 555.211,A -85,B 0,C 180,E1 -570.169,E2 -570.169} C_VEL
LIN {X 0,Y 601.332,Z 558.976,A -85,B 0,C 180,E1 -571.44,E2 -571.44} C_VEL
LIN {X 0,Y 601.333,Z 561.178,A -85,B 0,C 180,E1 -572.702,E2 -572.702} C_VEL
LIN {X 0,Y 601.324,Z 561.977,A -85,B 0,C 180,E1 -573.92,E2 -573.92} C_VEL
LIN {X 0,Y 601.32,Z 561.508,A -85,B 0,C 180,E1 -575.101,E2 -575.101} C_VEL
LIN {X 0,Y 601.318,Z 559.837,A -85,B 0,C 180,E1 -576.249,E2 -576.249} C_VEL
LIN {X 0,Y 601.336,Z 556.851,A -85,B 0,C 180,E1 -577.427,E2 -577.427} C_VEL
LIN {X 0,Y 601.331,Z 553.124,A -85,B 0,C 180,E1 -578.458,E2 -578.458} C_VEL
LIN {X 0,Y 601.357,Z 548.05,A -85,B 0,C 180,E1 -579.526,E2 -579.526} C_VEL
LIN {X 0,Y 601.384,Z 540.882,A -85,B 0,C 180,E1 -580.698,E2 -580.698} C_VEL
LIN {X 0,Y 601.39,Z 532.477,A -85,B 0,C 180,E1 -581.769,E2 -581.769} C_VEL
LIN {X 0,Y 601.431,Z 523.751,A -85,B 0,C 180,E1 -582.669,E2 -582.669} C_VEL
LIN {X 0,Y 601.467,Z 514.358,A -85,B 0,C 180,E1 -583.462,E2 -583.462} C_VEL
LIN {X 0,Y 601.476,Z 504.191,A -85,B 0,C 180,E1 -584.163,E2 -584.163} C_VEL
LIN {X 0,Y 601.515,Z 492.22,A -85,B 0,C 180,E1 -584.817,E2 -584.817} C_VEL
LIN {X 0,Y 601.579,Z 480.094,A -85,B 0,C 180,E1 -585.326,E2 -585.326} C_VEL
LIN {X 0,Y 601.429,Z 473.568,A -85,B 0,C 180,E1 -585.56,E2 -585.56} C_VEL
LIN {X 0,Y 601.411,Z 473.57,A -85,B 0,C 180,E1 -588.409,E2 -588.409} C_VEL
LIN {X 0,Y 601.414,Z 473.574,A -85,B 0,C 180,E1 -590.873,E2 -590.873} C_VEL
LIN {X 0,Y 601.385,Z 473.573,A -85,B 0,C 180,E1 -593.415,E2 -593.415} C_VEL
LIN {X 0,Y 601.438,Z 473.566,A -85,B 0,C 180,E1 -596.064,E2 -596.064} C_VEL
LIN {X 0,Y 601.421,Z 473.573,A -85,B 0,C 180,E1 -598.546,E2 -598.546} C_VEL
LIN {X 0,Y 601.431,Z 473.572,A -85,B 0,C 180,E1 -601.373,E2 -601.373} C_VEL
LIN {X 0,Y 601.404,Z 473.57,A -85,B 0,C 180,E1 -603.636,E2 -603.636} C_VEL
LIN {X 0,Y 601.391,Z 473.572,A -85,B 0,C 180,E1 -606.588,E2 -606.588} C_VEL
LIN {X 0,Y 601.429,Z 473.569,A -85,B 0,C 180,E1 -609.204,E2 -609.204} C_VEL
LIN {X 0,Y 601.386,Z 473.575,A -85,B 0,C 180,E1 -611.607,E2 -611.607} C_VEL
LIN {X 0,Y 601.417,Z 473.569,A -85,B 0,C 180,E1 -614.409,E2 -614.409} C_VEL
LIN {X 0,Y 601.408,Z 473.574,A -85,B 0,C 180,E1 -616.484,E2 -616.484} C_VEL
LIN {X 0,Y 601.417,Z 473.573,A -85,B 0,C 180,E1 -619.224,E2 -619.224} C_VEL
LIN {X 0,Y 601.445,Z 473.566,A -85,B 0,C 180,E1 -621.939,E2 -621.939} C_VEL
LIN {X 0,Y 601.409,Z 473.569,A -85,B 0,C 180,E1 -624.636,E2 -624.636} C_VEL
LIN {X 0,Y 601.431,Z 473.568,A -85,B 0,C 180,E1 -627.321,E2 -627.321} C_VEL
LIN {X 0,Y 601.449,Z 473.568,A -85,B 0,C 180,E1 -630,E2 -630} C_VEL
LIN {X 0,Y 601.441,Z 473.569,A -85,B 0,C 180,E1 -632.679,E2 -632.679} C_VEL
LIN {X 0,Y 601.405,Z 473.571,A -85,B 0,C 180,E1 -635.364,E2 -635.364} C_VEL
LIN {X 0,Y 601.446,Z 473.565,A -85,B 0,C 180,E1 -638.061,E2 -638.061} C_VEL
LIN {X 0,Y 601.399,Z 473.571,A -85,B 0,C 180,E1 -640.996,E2 -640.996} C_VEL
LIN {X 0,Y 601.423,Z 473.571,A -85,B 0,C 180,E1 -643.516,E2 -643.516} C_VEL
LIN {X 0,Y 601.427,Z 473.573,A -85,B 0,C 180,E1 -646.287,E2 -646.287} C_VEL
LIN {X 0,Y 601.417,Z 473.572,A -85,B 0,C 180,E1 -649.099,E2 -649.099} C_VEL
LIN {X 0,Y 601.406,Z 473.571,A -85,B 0,C 180,E1 -651.239,E2 -651.239} C_VEL
LIN {X 0,Y 601.436,Z 473.568,A -85,B 0,C 180,E1 -654.141,E2 -654.141} C_VEL
LIN {X 0,Y 601.427,Z 473.569,A -85,B 0,C 180,E1 -657.112,E2 -657.112} C_VEL
LIN {X 0,Y 601.402,Z 473.572,A -85,B 0,C 180,E1 -659.394,E2 -659.394} C_VEL
LIN {X 0,Y 601.406,Z 473.571,A -85,B 0,C 180,E1 -661.727,E2 -661.727} C_VEL
LIN {X 0,Y 601.417,Z 473.573,A -85,B 0,C 180,E1 -664.119,E2 -664.119} C_VEL
LIN {X 0,Y 601.398,Z 473.571,A -85,B 0,C 180,E1 -666.583,E2 -666.583} C_VEL
LIN {X 0,Y 601.406,Z 473.571,A -85,B 0,C 180,E1 -669.127,E2 -669.127} C_VEL
LIN {X 0,Y 601.421,Z 473.574,A -85,B 0,C 180,E1 -671.766,E2 -671.766} C_VEL
LIN {X 0,Y 601.455,Z 473.565,A -85,B 0,C 180,E1 -673.584,E2 -673.584} C_VEL
LIN {X 0,Y 601.409,Z 473.573,A -85,B 0,C 180,E1 -676.43,E2 -676.43} C_VEL
LIN {X 0,Y 601.41,Z 473.574,A -85,B 0,C 180,E1 -679.125,E2 -679.125} C_VEL
LIN {X 0,Y 601.415,Z 473.57,A -85,B 0,C 180,E1 -681.731,E2 -681.731} C_VEL
LIN {X 0,Y 601.389,Z 473.572,A -85,B 0,C 180,E1 -684.245,E2 -684.245} C_VEL
LIN {X 0,Y 601.427,Z 473.573,A -85,B 0,C 180,E1 -686.686,E2 -686.686} C_VEL
LIN {X 0,Y 601.405,Z 473.57,A -85,B 0,C 180,E1 -689.057,E2 -689.057} C_VEL
LIN {X 0,Y 601.435,Z 473.57,A -85,B 0,C 180,E1 -691.373,E2 -691.373} C_VEL
LIN {X 0,Y 601.405,Z 473.576,A -85,B 0,C 180,E1 -694.135,E2 -694.135} C_VEL
LIN {X 0,Y 601.398,Z 473.571,A -85,B 0,C 180,E1 -696.588,E2 -696.588} C_VEL
LIN {X 0,Y 601.416,Z 473.569,A -85,B 0,C 180,E1 -699.477,E2 -699.477} C_VEL
LIN {X 0,Y 601.393,Z 473.572,A -85,B 0,C 180,E1 -702.311,E2 -702.311} C_VEL
LIN {X 0,Y 601.415,Z 473.572,A -85,B 0,C 180,E1 -704.408,E2 -704.408} C_VEL
LIN {X 0,Y 601.404,Z 473.571,A -85,B 0,C 180,E1 -707.171,E2 -707.171} C_VEL
LIN {X 0,Y 601.437,Z 473.566,A -85,B 0,C 180,E1 -709.905,E2 -709.905} C_VEL
LIN {X 0,Y 601.398,Z 473.572,A -85,B 0,C 180,E1 -712.614,E2 -712.614} C_VEL
LIN {X 0,Y 601.42,Z 473.571,A -85,B 0,C 180,E1 -715.308,E2 -715.308} C_VEL
LIN {X 0,Y 601.435,Z 473.571,A -85,B 0,C 180,E1 -717.991,E2 -717.991} C_VEL
LIN {X 0,Y 601.442,Z 473.566,A -85,B 0,C 180,E1 -720.669,E2 -720.669} C_VEL
LIN {X 0,Y 601.377,Z 473.573,A -85,B 0,C 180,E1 -723.35,E2 -723.35} C_VEL
LIN {X 0,Y 601.416,Z 473.57,A -85,B 0,C 180,E1 -726.037,E2 -726.037} C_VEL
LIN {X 0,Y 601.412,Z 473.573,A -85,B 0,C 180,E1 -728.738,E2 -728.738} C_VEL
LIN {X 0,Y 601.412,Z 473.574,A -85,B 0,C 180,E1 -731.458,E2 -731.458} C_VEL
LIN {X 0,Y 601.423,Z 473.569,A -85,B 0,C 180,E1 -734.205,E2 -734.205} C_VEL
LIN {X 0,Y 601.404,Z 473.571,A -85,B 0,C 180,E1 -736.987,E2 -736.987} C_VEL
LIN {X 0,Y 601.408,Z 473.569,A -85,B 0,C 180,E1 -739.809,E2 -739.809} C_VEL
LIN {X 0,Y 601.402,Z 473.571,A -85,B 0,C 180,E1 -742.683,E2 -742.683} C_VEL
LIN {X 0,Y 601.402,Z 473.574,A -85,B 0,C 180,E1 -744.879,E2 -744.879} C_VEL
LIN {X 0,Y 601.384,Z 473.573,A -85,B 0,C 180,E1 -747.356,E2 -747.356} C_VEL
LIN {X 0,Y 601.432,Z 473.567,A -85,B 0,C 180,E1 -750.164,E2 -750.164} C_VEL
LIN {X 0,Y 601.419,Z 473.572,A -85,B 0,C 180,E1 -752.715,E2 -752.715} C_VEL
LIN {X 0,Y 601.379,Z 473.575,A -85,B 0,C 180,E1 -755.109,E2 -755.109} C_VEL
LIN {X 0,Y 601.437,Z 473.567,A -85,B 0,C 180,E1 -757.419,E2 -757.419} C_VEL
LIN {X 0,Y 601.403,Z 473.571,A -85,B 0,C 180,E1 -760.572,E2 -760.572} C_VEL
LIN {X 0,Y 601.412,Z 473.571,A -85,B 0,C 180,E1 -762.67,E2 -762.67} C_VEL
LIN {X 0,Y 601.4,Z 473.571,A -85,B 0,C 180,E1 -765.479,E2 -765.479} C_VEL
LIN {X 0,Y 601.426,Z 473.568,A -85,B 0,C 180,E1 -768.407,E2 -768.407} C_VEL
LIN {X 0,Y 601.392,Z 473.573,A -85,B 0,C 180,E1 -770.872,E2 -770.872} C_VEL
LIN {X 0,Y 601.418,Z 473.572,A -85,B 0,C 180,E1 -773.887,E2 -773.887} C_VEL
LIN {X 0,Y 601.474,Z 473.848,A -85,B 0,C 180,E1 -774.071,E2 -774.071} C_VEL
LIN {X 0,Y 601.708,Z 478.893,A -85,B 0,C 180,E1 -775.087,E2 -775.087} C_VEL
LIN {X 0,Y 601.813,Z 493.452,A -85,B 0,C 180,E1 -777.903,E2 -777.903} C_VEL
LIN {X 0,Y 601.703,Z 507.147,A -85,B 0,C 180,E1 -780.622,E2 -780.622} C_VEL
LIN {X 0,Y 601.624,Z 520.842,A -85,B 0,C 180,E1 -783.273,E2 -783.273} C_VEL
LIN {X 0,Y 601.58,Z 536.494,A -85,B 0,C 180,E1 -786.231,E2 -786.231} C_VEL
LIN {X 0,Y 601.506,Z 550.189,A -85,B 0,C 180,E1 -788.764,E2 -788.764} C_VEL
LIN {X 0,Y 601.479,Z 565.84,A -85,B 0,C 180,E1 -791.61,E2 -791.61} C_VEL
LIN {X 0,Y 601.453,Z 581.492,A -85,B 0,C 180,E1 -794.41,E2 -794.41} C_VEL
LIN {X 0,Y 601.379,Z 597.143,A -85,B 0,C 180,E1 -797.171,E2 -797.171} C_VEL
LIN {X 0,Y 601.415,Z 602.157,A -85,B 0,C 180,E1 -798.05,E2 -798.05} C_VEL
LIN {X 0,Y 601.592,Z 614.44,A -85,B 0,C 180,E1 -798.267,E2 -798.267} C_VEL
LIN {X 0,Y 601.561,Z 627.258,A -85,B 0,C 180,E1 -798.623,E2 -798.623} C_VEL
LIN {X 0,Y 601.531,Z 639.047,A -85,B 0,C 180,E1 -799.08,E2 -799.08} C_VEL
LIN {X 0,Y 601.482,Z 650.328,A -85,B 0,C 180,E1 -799.651,E2 -799.651} C_VEL
LIN {X 0,Y 601.469,Z 660.931,A -85,B 0,C 180,E1 -800.33,E2 -800.33} C_VEL
LIN {X 0,Y 601.435,Z 670.599,A -85,B 0,C 180,E1 -801.093,E2 -801.093} C_VEL
LIN {X 0,Y 601.407,Z 679.414,A -85,B 0,C 180,E1 -801.939,E2 -801.939} C_VEL
LIN {X 0,Y 601.388,Z 686.691,A -85,B 0,C 180,E1 -802.783,E2 -802.783} C_VEL
LIN {X 0,Y 601.375,Z 693.773,A -85,B 0,C 180,E1 -803.782,E2 -803.782} C_VEL
LIN {X 0,Y 601.373,Z 698.68,A -85,B 0,C 180,E1 -804.635,E2 -804.635} C_VEL
LIN {X 0,Y 601.354,Z 703.371,A -85,B 0,C 180,E1 -805.643,E2 -805.643} C_VEL
LIN {X 0,Y 601.344,Z 706.956,A -85,B 0,C 180,E1 -806.65,E2 -806.65} C_VEL
LIN {X 0,Y 601.325,Z 708.809,A -85,B 0,C 180,E1 -807.321,E2 -807.321} C_VEL
LIN {X 0,Y 601.343,Z 710.202,A -85,B 0,C 180,E1 -807.991,E2 -807.991} C_VEL
LIN {X 0,Y 601.339,Z 711.784,A -85,B 0,C 180,E1 -809.33,E2 -809.33} C_VEL
LIN {X 0,Y 601.335,Z 712,A -85,B 0,C 180,E1 -810,E2 -810} C_VEL
LIN {X 0,Y 601.347,Z 711.184,A -85,B 0,C 180,E1 -811.339,E2 -811.339} C_VEL
LIN {X 0,Y 601.343,Z 710.202,A -85,B 0,C 180,E1 -812.009,E2 -812.009} C_VEL
LIN {X 0,Y 601.325,Z 708.809,A -85,B 0,C 180,E1 -812.68,E2 -812.68} C_VEL
LIN {X 0,Y 601.368,Z 705.896,A -85,B 0,C 180,E1 -813.685,E2 -813.685} C_VEL
LIN {X 0,Y 601.336,Z 701.949,A -85,B 0,C 180,E1 -814.693,E2 -814.693} C_VEL
LIN {X 0,Y 601.372,Z 695.876,A -85,B 0,C 180,E1 -815.869,E2 -815.869} C_VEL
LIN {X 0,Y 601.382,Z 689.234,A -85,B 0,C 180,E1 -816.88,E2 -816.88} C_VEL
LIN {X 0,Y 601.401,Z 680.988,A -85,B 0,C 180,E1 -817.892,E2 -817.892} C_VEL
LIN {X 0,Y 601.436,Z 672.535,A -85,B 0,C 180,E1 -818.738,E2 -818.738} C_VEL
LIN {X 0,Y 601.45,Z 662.09,A -85,B 0,C 180,E1 -819.585,E2 -819.585} C_VEL
LIN {X 0,Y 601.481,Z 651.754,A -85,B 0,C 180,E1 -820.264,E2 -820.264} C_VEL
LIN {X 0,Y 601.512,Z 639.9,A -85,B 0,C 180,E1 -820.883,E2 -820.883} C_VEL
LIN {X 0,Y 601.561,Z 627.269,A -85,B 0,C 180,E1 -821.377,E2 -821.377} C_VEL
LIN {X 0,Y 601.592,Z 614.431,A -85,B 0,C 180,E1 -821.733,E2 -821.733} C_VEL
LIN {X 0,Y 601.416,Z 602.156,A -85,B 0,C 180,E1 -821.95,E2 -821.95} C_VEL
LIN {X 0,Y 601.402,Z 587.36,A -85,B 0,C 180,E1 -824.552,E2 -824.552} C_VEL
LIN {X 0,Y 601.468,Z 571.709,A -85,B 0,C 180,E1 -827.335,E2 -827.335} C_VEL
LIN {X 0,Y 601.48,Z 556.057,A -85,B 0,C 180,E1 -830.163,E2 -830.163} C_VEL
LIN {X 0,Y 601.58,Z 540.406,A -85,B 0,C 180,E1 -833.04,E2 -833.04} C_VEL
LIN {X 0,Y 601.633,Z 525.124,A -85,B 0,C 180,E1 -835.91,E2 -835.91} C_VEL
LIN {X 0,Y 601.687,Z 511.059,A -85,B 0,C 180,E1 -838.614,E2 -838.614} C_VEL
LIN {X 0,Y 601.727,Z 497.868,A -85,B 0,C 180,E1 -841.215,E2 -841.215} C_VEL
LIN {X 0,Y 601.717,Z 489.948,A -85,B 0,C 180,E1 -842.759,E2 -842.759} C_VEL
LIN {X 0,Y 601.64,Z 475.803,A -85,B 0,C 180,E1 -845.399,E2 -845.399} C_VEL
LIN {X 0,Y 601.43,Z 473.572,A -85,B 0,C 180,E1 -845.842,E2 -845.842} C_VEL
LIN {X 0,Y 601.434,Z 473.57,A -85,B 0,C 180,E1 -848.471,E2 -848.471} C_VEL
LIN {X 0,Y 601.427,Z 473.57,A -85,B 0,C 180,E1 -851.593,E2 -851.593} C_VEL
LIN {X 0,Y 601.429,Z 473.57,A -85,B 0,C 180,E1 -854.535,E2 -854.535} C_VEL
LIN {X 0,Y 601.413,Z 473.575,A -85,B 0,C 180,E1 -857.41,E2 -857.41} C_VEL
LIN {X 0,Y 601.404,Z 473.575,A -85,B 0,C 180,E1 -860.004,E2 -860.004} C_VEL
LIN {X 0,Y 601.434,Z 473.57,A -85,B 0,C 180,E1 -862.619,E2 -862.619} C_VEL
LIN {X 0,Y 601.405,Z 473.574,A -85,B 0,C 180,E1 -865.067,E2 -865.067} C_VEL
LIN {X 0,Y 601.436,Z 473.571,A -85,B 0,C 180,E1 -867.485,E2 -867.485} C_VEL
LIN {X 0,Y 601.432,Z 473.573,A -85,B 0,C 180,E1 -869.852,E2 -869.852} C_VEL
LIN {X 0,Y 601.407,Z 473.573,A -85,B 0,C 180,E1 -872.64,E2 -872.64} C_VEL
LIN {X 0,Y 601.4,Z 473.574,A -85,B 0,C 180,E1 -875.121,E2 -875.121} C_VEL
LIN {X 0,Y 601.42,Z 473.574,A -85,B 0,C 180,E1 -877.395,E2 -877.395} C_VEL
LIN {X 0,Y 601.403,Z 473.573,A -85,B 0,C 180,E1 -880.191,E2 -880.191} C_VEL
LIN {X 0,Y 601.413,Z 473.571,A -85,B 0,C 180,E1 -883.014,E2 -883.014} C_VEL
LIN {X 0,Y 601.424,Z 473.572,A -85,B 0,C 180,E1 -885.909,E2 -885.909} C_VEL
LIN {X 0,Y 601.418,Z 473.574,A -85,B 0,C 180,E1 -888.542,E2 -888.542} C_VEL
LIN {X 0,Y 601.411,Z 473.573,A -85,B 0,C 180,E1 -891.262,E2 -891.262} C_VEL
LIN {X 0,Y 601.42,Z 473.57,A -85,B 0,C 180,E1 -893.963,E2 -893.963} C_VEL
LIN {X 0,Y 601.388,Z 473.574,A -85,B 0,C 180,E1 -896.65,E2 -896.65} C_VEL
LIN {X 0,Y 601.439,Z 473.568,A -85,B 0,C 180,E1 -899.331,E2 -899.331} C_VEL
LIN {X 0,Y 601.434,Z 473.57,A -85,B 0,C 180,E1 -902.009,E2 -902.009} C_VEL
LIN {X 0,Y 601.425,Z 473.574,A -85,B 0,C 180,E1 -904.692,E2 -904.692} C_VEL
LIN {X 0,Y 601.446,Z 473.569,A -85,B 0,C 180,E1 -907.385,E2 -907.385} C_VEL
LIN {X 0,Y 601.439,Z 473.568,A -85,B 0,C 180,E1 -910.095,E2 -910.095} C_VEL
LIN {X 0,Y 601.405,Z 473.573,A -85,B 0,C 180,E1 -912.354,E2 -912.354} C_VEL
LIN {X 0,Y 600.736,Z 473.656,A -85,B 0,C 180,E1 -912.914,E2 -912.914} C_VEL
LIN {X 0,Y 597.888,Z 474.011,A -85,B 0,C 180,E1 -913.822,E2 -913.822} C_VEL
LIN {X 0,Y 595.482,Z 474.313,A -85,B 0,C 180,E1 -914.552,E2 -914.552} C_VEL
LIN {X 0,Y 594.444,Z 474.44,A -85,B 0,C 180,E1 -915.116,E2 -915.116} C_VEL
LIN {X 0,Y 594.357,Z 474.45,A -85,B 0,C 180,E1 -915.307,E2 -915.307} C_VEL
LIN {X 0,Y 594.358,Z 474.45,A -85,B 0,C 180,E1 -917.905,E2 -917.905} C_VEL
LIN {X 0,Y 594.391,Z 474.45,A -85,B 0,C 180,E1 -920.918,E2 -920.918} C_VEL
LIN {X 0,Y 594.399,Z 474.511,A -85,B 0,C 180,E1 -922.438,E2 -922.438} C_VEL
LIN {X 0,Y 594.561,Z 486.087,A -85,B 0,C 180,E1 -922.868,E2 -922.868} C_VEL
LIN {X 0,Y 594.516,Z 497.573,A -85,B 0,C 180,E1 -923.422,E2 -923.422} C_VEL
LIN {X 0,Y 594.441,Z 508.239,A -85,B 0,C 180,E1 -924.073,E2 -924.073} C_VEL
LIN {X 0,Y 594.416,Z 519.235,A -85,B 0,C 180,E1 -924.911,E2 -924.911} C_VEL
LIN {X 0,Y 594.351,Z 528.178,A -85,B 0,C 180,E1 -925.757,E2 -925.757} C_VEL
LIN {X 0,Y 594.321,Z 536.38,A -85,B 0,C 180,E1 -926.703,E2 -926.703} C_VEL
LIN {X 0,Y 594.298,Z 543.012,A -85,B 0,C 180,E1 -927.637,E2 -927.637} C_VEL
LIN {X 0,Y 594.258,Z 548.504,A -85,B 0,C 180,E1 -928.585,E2 -928.585} C_VEL
LIN {X 0,Y 594.276,Z 553.964,A -85,B 0,C 180,E1 -929.782,E2 -929.782} C_VEL
LIN {X 0,Y 594.243,Z 557.847,A -85,B 0,C 180,E1 -930.962,E2 -930.962} C_VEL
LIN {X 0,Y 594.211,Z 560.439,A -85,B 0,C 180,E1 -932.157,E2 -932.157} C_VEL
LIN {X 0,Y 594.249,Z 561.49,A -85,B 0,C 180,E1 -932.959,E2 -932.959} C_VEL
LIN {X 0,Y 594.246,Z 561.989,A -85,B 0,C 180,E1 -934.119,E2 -934.119} C_VEL
LIN {X 0,Y 594.225,Z 561.162,A -85,B 0,C 180,E1 -935.418,E2 -935.418} C_VEL
LIN {X 0,Y 594.224,Z 559.442,A -85,B 0,C 180,E1 -936.462,E2 -936.462} C_VEL
LIN {X 0,Y 594.24,Z 556.468,A -85,B 0,C 180,E1 -937.589,E2 -937.589} C_VEL
LIN {X 0,Y 594.272,Z 551.85,A -85,B 0,C 180,E1 -938.814,E2 -938.814} C_VEL
LIN {X 0,Y 594.281,Z 546.212,A -85,B 0,C 180,E1 -939.929,E2 -939.929} C_VEL
LIN {X 0,Y 594.301,Z 538.444,A -85,B 0,C 180,E1 -941.117,E2 -941.117} C_VEL
LIN {X 0,Y 594.365,Z 530.526,A -85,B 0,C 180,E1 -942.081,E2 -942.081} C_VEL
LIN {X 0,Y 594.39,Z 522.264,A -85,B 0,C 180,E1 -942.91,E2 -942.91} C_VEL
LIN {X 0,Y 594.447,Z 512.317,A -85,B 0,C 180,E1 -943.728,E2 -943.728} C_VEL
LIN {X 0,Y 594.499,Z 500.412,A -85,B 0,C 180,E1 -944.512,E2 -944.512} C_VEL
LIN {X 0,Y 594.556,Z 488.533,A -85,B 0,C 180,E1 -945.115,E2 -945.115} C_VEL
LIN {X 0,Y 594.593,Z 477.255,A -85,B 0,C 180,E1 -945.556,E2 -945.556} C_VEL
LIN {X 0,Y 594.391,Z 474.444,A -85,B 0,C 180,E1 -945.665,E2 -945.665} C_VEL
LIN {X 0,Y 594.37,Z 474.447,A -85,B 0,C 180,E1 -948.535,E2 -948.535} C_VEL
LIN {X 0,Y 594.381,Z 474.447,A -85,B 0,C 180,E1 -951.297,E2 -951.297} C_VEL
LIN {X 0,Y 594.348,Z 474.453,A -85,B 0,C 180,E1 -953.755,E2 -953.755} C_VEL
LIN {X 0,Y 594.381,Z 474.445,A -85,B 0,C 180,E1 -956.239,E2 -956.239} C_VEL
LIN {X 0,Y 594.368,Z 474.45,A -85,B 0,C 180,E1 -958.649,E2 -958.649} C_VEL
LIN {X 0,Y 594.383,Z 474.446,A -85,B 0,C 180,E1 -961.043,E2 -961.043} C_VEL
LIN {X 0,Y 594.389,Z 474.446,A -85,B 0,C 180,E1 -963.3,E2 -963.3} C_VEL
LIN {X 0,Y 594.367,Z 474.448,A -85,B 0,C 180,E1 -966.295,E2 -966.295} C_VEL
LIN {X 0,Y 594.398,Z 474.445,A -85,B 0,C 180,E1 -969.224,E2 -969.224} C_VEL
LIN {X 0,Y 594.336,Z 474.454,A -85,B 0,C 180,E1 -972.094,E2 -972.094} C_VEL
LIN {X 0,Y 594.371,Z 474.446,A -85,B 0,C 180,E1 -974.219,E2 -974.219} C_VEL
LIN {X 0,Y 594.378,Z 474.451,A -85,B 0,C 180,E1 -976.321,E2 -976.321} C_VEL
LIN {X 0,Y 594.376,Z 474.448,A -85,B 0,C 180,E1 -979.095,E2 -979.095} C_VEL
LIN {X 0,Y 594.389,Z 474.445,A -85,B 0,C 180,E1 -981.843,E2 -981.843} C_VEL
LIN {X 0,Y 594.376,Z 474.446,A -85,B 0,C 180,E1 -984.572,E2 -984.572} C_VEL
LIN {X 0,Y 594.399,Z 474.444,A -85,B 0,C 180,E1 -987.289,E2 -987.289} C_VEL
LIN {X 0,Y 594.418,Z 474.444,A -85,B 0,C 180,E1 -990,E2 -990} C_VEL
LIN {X 0,Y 594.407,Z 474.446,A -85,B 0,C 180,E1 -992.711,E2 -992.711} C_VEL
LIN {X 0,Y 594.374,Z 474.447,A -85,B 0,C 180,E1 -995.428,E2 -995.428} C_VEL
LIN {X 0,Y 594.418,Z 474.44,A -85,B 0,C 180,E1 -998.157,E2 -998.157} C_VEL
LIN {X 0,Y 594.37,Z 474.446,A -85,B 0,C 180,E1 -1001.061,E2 -1001.061} C_VEL
LIN {X 0,Y 594.388,Z 474.446,A -85,B 0,C 180,E1 -1003.679,E2 -1003.679} C_VEL
LIN {X 0,Y 594.382,Z 474.449,A -85,B 0,C 180,E1 -1006.486,E2 -1006.486} C_VEL
LIN {X 0,Y 594.37,Z 474.452,A -85,B 0,C 180,E1 -1009.334,E2 -1009.334} C_VEL
LIN {X 0,Y 594.365,Z 474.447,A -85,B 0,C 180,E1 -1011.503,E2 -1011.503} C_VEL
LIN {X 0,Y 594.373,Z 474.446,A -85,B 0,C 180,E1 -1014.447,E2 -1014.447} C_VEL
LIN {X 0,Y 594.375,Z 474.451,A -85,B 0,C 180,E1 -1016.7,E2 -1016.7} C_VEL
LIN {X 0,Y 594.377,Z 474.446,A -85,B 0,C 180,E1 -1018.999,E2 -1018.999} C_VEL
LIN {X 0,Y 594.382,Z 474.446,A -85,B 0,C 180,E1 -1021.642,E2 -1021.642} C_VEL
LIN {X 0,Y 594.365,Z 474.449,A -85,B 0,C 180,E1 -1024.581,E2 -1024.581} C_VEL
LIN {X 0,Y 594.394,Z 474.445,A -85,B 0,C 180,E1 -1027.608,E2 -1027.608} C_VEL
LIN {X 0,Y 594.362,Z 474.449,A -85,B 0,C 180,E1 -1030.568,E2 -1030.568} C_VEL
LIN {X 0,Y 594.379,Z 474.45,A -85,B 0,C 180,E1 -1033.299,E2 -1033.299} C_VEL
LIN {X 0,Y 594.348,Z 474.455,A -85,B 0,C 180,E1 -1036.163,E2 -1036.163} C_VEL
LIN {X 0,Y 594.378,Z 474.445,A -85,B 0,C 180,E1 -1038.535,E2 -1038.535} C_VEL
LIN {X 0,Y 594.374,Z 474.446,A -85,B 0,C 180,E1 -1041.297,E2 -1041.297} C_VEL
LIN {X 0,Y 594.35,Z 474.454,A -85,B 0,C 180,E1 -1043.755,E2 -1043.755} C_VEL
LIN {X 0,Y 594.382,Z 474.446,A -85,B 0,C 180,E1 -1046.239,E2 -1046.239} C_VEL
LIN {X 0,Y 594.364,Z 474.448,A -85,B 0,C 180,E1 -1048.649,E2 -1048.649} C_VEL
LIN {X 0,Y 594.387,Z 474.448,A -85,B 0,C 180,E1 -1051.042,E2 -1051.042} C_VEL
LIN {X 0,Y 594.369,Z 474.447,A -85,B 0,C 180,E1 -1053.299,E2 -1053.299} C_VEL
LIN {X 0,Y 594.381,Z 474.445,A -85,B 0,C 180,E1 -1056.295,E2 -1056.295} C_VEL
LIN {X 0,Y 594.391,Z 474.444,A -85,B 0,C 180,E1 -1059.224,E2 -1059.224} C_VEL
LIN {X 0,Y 594.349,Z 474.45,A -85,B 0,C 180,E1 -1062.095,E2 -1062.095} C_VEL
LIN {X 0,Y 594.369,Z 474.448,A -85,B 0,C 180,E1 -1064.219,E2 -1064.219} C_VEL
LIN {X 0,Y 594.373,Z 474.45,A -85,B 0,C 180,E1 -1066.321,E2 -1066.321} C_VEL
LIN {X 0,Y 594.378,Z 474.451,A -85,B 0,C 180,E1 -1069.094,E2 -1069.094} C_VEL
LIN {X 0,Y 594.382,Z 474.447,A -85,B 0,C 180,E1 -1071.843,E2 -1071.843} C_VEL
LIN {X 0,Y 594.387,Z 474.445,A -85,B 0,C 180,E1 -1074.572,E2 -1074.572} C_VEL
LIN {X 0,Y 594.387,Z 474.444,A -85,B 0,C 180,E1 -1077.289,E2 -1077.289} C_VEL
LIN {X 0,Y 594.418,Z 474.442,A -85,B 0,C 180,E1 -1080,E2 -1080} C_VEL
LIN {X 0,Y 594.406,Z 474.446,A -85,B 0,C 180,E1 -1082.711,E2 -1082.711} C_VEL
LIN {X 0,Y 594.38,Z 474.449,A -85,B 0,C 180,E1 -1085.428,E2 -1085.428} C_VEL
LIN {X 0,Y 594.416,Z 474.442,A -85,B 0,C 180,E1 -1088.157,E2 -1088.157} C_VEL
LIN {X 0,Y 594.374,Z 474.447,A -85,B 0,C 180,E1 -1091.064,E2 -1091.064} C_VEL
LIN {X 0,Y 594.386,Z 474.444,A -85,B 0,C 180,E1 -1093.679,E2 -1093.679} C_VEL
LIN {X 0,Y 594.366,Z 474.448,A -85,B 0,C 180,E1 -1096.486,E2 -1096.486} C_VEL
LIN {X 0,Y 594.369,Z 474.449,A -85,B 0,C 180,E1 -1099.334,E2 -1099.334} C_VEL
LIN {X 0,Y 594.352,Z 474.449,A -85,B 0,C 180,E1 -1101.504,E2 -1101.504} C_VEL
LIN {X 0,Y 594.392,Z 474.444,A -85,B 0,C 180,E1 -1104.446,E2 -1104.446} C_VEL
LIN {X 0,Y 594.358,Z 474.452,A -85,B 0,C 180,E1 -1106.701,E2 -1106.701} C_VEL
LIN {X 0,Y 594.374,Z 474.447,A -85,B 0,C 180,E1 -1108.999,E2 -1108.999} C_VEL
LIN {X 0,Y 594.38,Z 474.445,A -85,B 0,C 180,E1 -1111.643,E2 -1111.643} C_VEL
LIN {X 0,Y 594.361,Z 474.448,A -85,B 0,C 180,E1 -1114.581,E2 -1114.581} C_VEL
LIN {X 0,Y 594.392,Z 474.444,A -85,B 0,C 180,E1 -1117.608,E2 -1117.608} C_VEL
LIN {X 0,Y 594.358,Z 474.448,A -85,B 0,C 180,E1 -1120.568,E2 -1120.568} C_VEL
LIN {X 0,Y 594.368,Z 474.448,A -85,B 0,C 180,E1 -1123.299,E2 -1123.299} C_VEL
LIN {X 0,Y 594.345,Z 474.453,A -85,B 0,C 180,E1 -1126.163,E2 -1126.163} C_VEL
LIN {X 0,Y 594.383,Z 474.445,A -85,B 0,C 180,E1 -1128.536,E2 -1128.536} C_VEL
LIN {X 0,Y 594.367,Z 474.447,A -85,B 0,C 180,E1 -1131.298,E2 -1131.298} C_VEL
LIN {X 0,Y 594.395,Z 474.543,A -85,B 0,C 180,E1 -1133.811,E2 -1133.811} C_VEL
LIN {X 0,Y 594.844,Z 478.446,A -85,B 0,C 180,E1 -1134.625,E2 -1134.625} C_VEL
LIN {X 0,Y 594.803,Z 491.862,A -85,B 0,C 180,E1 -1137.278,E2 -1137.278} C_VEL
LIN {X 0,Y 594.868,Z 503.858,A -85,B 0,C 180,E1 -1139.593,E2 -1139.593} C_VEL
LIN {X 0,Y 594.76,Z 518.099,A -85,B 0,C 180,E1 -1142.405,E2 -1142.405} C_VEL
LIN {X 0,Y 594.639,Z 530.625,A -85,B 0,C 180,E1 -1144.819,E2 -1144.819} C_VEL
LIN {X 0,Y 594.594,Z 544.748,A -85,B 0,C 180,E1 -1147.49,E2 -1147.49} C_VEL
LIN {X 0,Y 594.493,Z 559.971,A -85,B 0,C 180,E1 -1150.311,E2 -1150.311} C_VEL
LIN {X 0,Y 594.436,Z 575.248,A -85,B 0,C 180,E1 -1153.095,E2 -1153.095} C_VEL
LIN {X 0,Y 594.387,Z 591.866,A -85,B 0,C 180,E1 -1156.078,E2 -1156.078} C_VEL
LIN {X 0,Y 594.359,Z 602.157,A -85,B 0,C 180,E1 -1157.906,E2 -1157.906} C_VEL
LIN {X 0,Y 594.675,Z 607.948,A -85,B 0,C 180,E1 -1157.999,E2 -1157.999} C_VEL
LIN {X 0,Y 594.623,Z 621.218,A -85,B 0,C 180,E1 -1158.301,E2 -1158.301} C_VEL
LIN {X 0,Y 594.561,Z 634.305,A -85,B 0,C 180,E1 -1158.746,E2 -1158.746} C_VEL
LIN {X 0,Y 594.518,Z 645.634,A -85,B 0,C 180,E1 -1159.27,E2 -1159.27} C_VEL
LIN {X 0,Y 594.481,Z 657.2,A -85,B 0,C 180,E1 -1159.958,E2 -1159.958} C_VEL
LIN {X 0,Y 594.414,Z 667.596,A -85,B 0,C 180,E1 -1160.73,E2 -1160.73} C_VEL
LIN {X 0,Y 594.383,Z 676.112,A -85,B 0,C 180,E1 -1161.501,E2 -1161.501} C_VEL
LIN {X 0,Y 594.347,Z 683.961,A -85,B 0,C 180,E1 -1162.355,E2 -1162.355} C_VEL
LIN {X 0,Y 594.282,Z 691.812,A -85,B 0,C 180,E1 -1163.408,E2 -1163.408} C_VEL
LIN {X 0,Y 594.289,Z 698.681,A -85,B 0,C 180,E1 -1164.571,E2 -1164.571} C_VEL
LIN {X 0,Y 594.27,Z 703.371,A -85,B 0,C 180,E1 -1165.591,E2 -1165.591} C_VEL
LIN {X 0,Y 594.267,Z 706.956,A -85,B 0,C 180,E1 -1166.61,E2 -1166.61} C_VEL
LIN {X 0,Y 594.225,Z 708.809,A -85,B 0,C 180,E1 -1167.288,E2 -1167.288} C_VEL
LIN {X 0,Y 594.241,Z 710.202,A -85,B 0,C 180,E1 -1167.967,E2 -1167.967} C_VEL
LIN {X 0,Y 594.239,Z 711.784,A -85,B 0,C 180,E1 -1169.322,E2 -1169.322} C_VEL
LIN {X 0,Y 594.236,Z 712,A -85,B 0,C 180,E1 -1170,E2 -1170} C_VEL
LIN {X 0,Y 594.247,Z 711.184,A -85,B 0,C 180,E1 -1171.355,E2 -1171.355} C_VEL
LIN {X 0,Y 594.241,Z 710.202,A -85,B 0,C 180,E1 -1172.033,E2 -1172.033} C_VEL
LIN {X 0,Y 594.226,Z 708.809,A -85,B 0,C 180,E1 -1172.712,E2 -1172.712} C_VEL
LIN {X 0,Y 594.289,Z 705.896,A -85,B 0,C 180,E1 -1173.729,E2 -1173.729} C_VEL
LIN {X 0,Y 594.241,Z 701.949,A -85,B 0,C 180,E1 -1174.749,E2 -1174.749} C_VEL
LIN {X 0,Y 594.304,Z 695.876,A -85,B 0,C 180,E1 -1175.939,E2 -1175.939} C_VEL
LIN {X 0,Y 594.308,Z 689.235,A -85,B 0,C 180,E1 -1176.962,E2 -1176.962} C_VEL
LIN {X 0,Y 594.359,Z 680.988,A -85,B 0,C 180,E1 -1177.987,E2 -1177.987} C_VEL
LIN {X 0,Y 594.382,Z 672.535,A -85,B 0,C 180,E1 -1178.842,E2 -1178.842} C_VEL
LIN {X 0,Y 594.433,Z 662.091,A -85,B 0,C 180,E1 -1179.699,E2 -1179.699} C_VEL
LIN {X 0,Y 594.481,Z 651.755,A -85,B 0,C 180,E1 -1180.387,E2 -1180.387} C_VEL
LIN {X 0,Y 594.527,Z 640.816,A -85,B 0,C 180,E1 -1180.969,E2 -1180.969} C_VEL
LIN {X 0,Y 594.593,Z 628.734,A -85,B 0,C 180,E1 -1181.463,E2 -1181.463} C_VEL
LIN {X 0,Y 594.631,Z 615.344,A -85,B 0,C 180,E1 -1181.851,E2 -1181.851} C_VEL
LIN {X 0,Y 594.58,Z 603.59,A -85,B 0,C 180,E1 -1182.068,E2 -1182.068} C_VEL
LIN {X 0,Y 594.364,Z 602.033,A -85,B 0,C 180,E1 -1182.116,E2 -1182.116} C_VEL
LIN {X 0,Y 594.369,Z 587.36,A -85,B 0,C 180,E1 -1184.728,E2 -1184.728} C_VEL
LIN {X 0,Y 594.462,Z 571.709,A -85,B 0,C 180,E1 -1187.546,E2 -1187.546} C_VEL
LIN {X 0,Y 594.499,Z 556.057,A -85,B 0,C 180,E1 -1190.411,E2 -1190.411} C_VEL
LIN {X 0,Y 594.615,Z 542.362,A -85,B 0,C 180,E1 -1192.957,E2 -1192.957} C_VEL
LIN {X 0,Y 594.662,Z 528.667,A -85,B 0,C 180,E1 -1195.555,E2 -1195.555} C_VEL
LIN {X 0,Y 594.775,Z 514.972,A -85,B 0,C 180,E1 -1198.207,E2 -1198.207} C_VEL
LIN {X 0,Y 594.87,Z 501.277,A -85,B 0,C 180,E1 -1200.926,E2 -1200.926} C_VEL
LIN {X 0,Y 594.738,Z 487.257,A -85,B 0,C 180,E1 -1203.535,E2 -1203.535} C_VEL
LIN {X 0,Y 594.573,Z 475.408,A -85,B 0,C 180,E1 -1205.811,E2 -1205.811} C_VEL
LIN {X 0,Y 594.374,Z 474.452,A -85,B 0,C 180,E1 -1206.034,E2 -1206.034} C_VEL
LIN {X 0,Y 594.378,Z 474.451,A -85,B 0,C 180,E1 -1208.806,E2 -1208.806} C_VEL
LIN {X 0,Y 594.388,Z 474.446,A -85,B 0,C 180,E1 -1211.849,E2 -1211.849} C_VEL
LIN {X 0,Y 594.368,Z 474.452,A -85,B 0,C 180,E1 -1214.809,E2 -1214.809} C_VEL
LIN {X 0,Y 594.371,Z 474.451,A -85,B 0,C 180,E1 -1217.625,E2 -1217.625} C_VEL
LIN {X 0,Y 594.372,Z 474.449,A -85,B 0,C 180,E1 -1220.319,E2 -1220.319} C_VEL
LIN {X 0,Y 594.38,Z 474.447,A -85,B 0,C 180,E1 -1222.913,E2 -1222.913} C_VEL
LIN {X 0,Y 594.373,Z 474.449,A -85,B 0,C 180,E1 -1225.863,E2 -1225.863} C_VEL
LIN {X 0,Y 594.372,Z 474.452,A -85,B 0,C 180,E1 -1228.65,E2 -1228.65} C_VEL
LIN {X 0,Y 594.386,Z 474.449,A -85,B 0,C 180,E1 -1231.043,E2 -1231.043} C_VEL
LIN {X 0,Y 594.386,Z 474.447,A -85,B 0,C 180,E1 -1233.978,E2 -1233.978} C_VEL
LIN {X 0,Y 594.378,Z 474.449,A -85,B 0,C 180,E1 -1236.296,E2 -1236.296} C_VEL
LIN {X 0,Y 594.394,Z 474.445,A -85,B 0,C 180,E1 -1239.224,E2 -1239.224} C_VEL
LIN {X 0,Y 594.353,Z 474.452,A -85,B 0,C 180,E1 -1242.095,E2 -1242.095} C_VEL
LIN {X 0,Y 594.373,Z 474.448,A -85,B 0,C 180,E1 -1244.219,E2 -1244.219} C_VEL
LIN {X 0,Y 594.364,Z 474.45,A -85,B 0,C 180,E1 -1247.017,E2 -1247.017} C_VEL
LIN {X 0,Y 594.389,Z 474.45,A -85,B 0,C 180,E1 -1249.784,E2 -1249.784} C_VEL
LIN {X 0,Y 594.373,Z 474.449,A -85,B 0,C 180,E1 -1252.527,E2 -1252.527} C_VEL
LIN {X 0,Y 594.38,Z 474.447,A -85,B 0,C 180,E1 -1255.252,E2 -1255.252} C_VEL
LIN {X 0,Y 594.406,Z 474.444,A -85,B 0,C 180,E1 -1257.967,E2 -1257.967} C_VEL
LIN {X 0,Y 594.42,Z 474.443,A -85,B 0,C 180,E1 -1260.678,E2 -1260.678} C_VEL
LIN {X 0,Y 594.379,Z 474.451,A -85,B 0,C 180,E1 -1263.39,E2 -1263.39} C_VEL
LIN {X 0,Y 594.363,Z 474.451,A -85,B 0,C 180,E1 -1266.109,E2 -1266.109} C_VEL
LIN {X 0,Y 594.379,Z 474.447,A -85,B 0,C 180,E1 -1268.842,E2 -1268.842} C_VEL
LIN {X 0,Y 594.385,Z 474.446,A -85,B 0,C 180,E1 -1271.596,E2 -1271.596} C_VEL
LIN {X 0,Y 594.394,Z 474.447,A -85,B 0,C 180,E1 -1274.377,E2 -1274.377} C_VEL
LIN {X 0,Y 594.357,Z 474.45,A -85,B 0,C 180,E1 -1275.307,E2 -1275.307} C_VEL
LIN {X 0,Y 593.681,Z 474.538,A -85,B 0,C 180,E1 -1275.872,E2 -1275.872} C_VEL
LIN {X 0,Y 590.82,Z 474.894,A -85,B 0,C 180,E1 -1276.79,E2 -1276.79} C_VEL
LIN {X 0,Y 588.414,Z 475.194,A -85,B 0,C 180,E1 -1277.529,E2 -1277.529} C_VEL
LIN {X 0,Y 587.391,Z 475.32,A -85,B 0,C 180,E1 -1278.099,E2 -1278.099} C_VEL
LIN {X 0,Y 587.313,Z 475.328,A -85,B 0,C 180,E1 -1278.292,E2 -1278.292} C_VEL
LIN {X 0,Y 587.337,Z 475.327,A -85,B 0,C 180,E1 -1281.038,E2 -1281.038} C_VEL
LIN {X 0,Y 587.35,Z 475.419,A -85,B 0,C 180,E1 -1282.328,E2 -1282.328} C_VEL
LIN {X 0,Y 587.607,Z 483.377,A -85,B 0,C 180,E1 -1282.619,E2 -1282.619} C_VEL
LIN {X 0,Y 587.539,Z 494.853,A -85,B 0,C 180,E1 -1283.146,E2 -1283.146} C_VEL
LIN {X 0,Y 587.461,Z 506.174,A -85,B 0,C 180,E1 -1283.814,E2 -1283.814} C_VEL
LIN {X 0,Y 587.391,Z 516.67,A -85,B 0,C 180,E1 -1284.587,E2 -1284.587} C_VEL
LIN {X 0,Y 587.299,Z 526.876,A -85,B 0,C 180,E1 -1285.519,E2 -1285.519} C_VEL
LIN {X 0,Y 587.27,Z 535.273,A -85,B 0,C 180,E1 -1286.474,E2 -1286.474} C_VEL
LIN {X 0,Y 587.224,Z 541.712,A -85,B 0,C 180,E1 -1287.359,E2 -1287.359} C_VEL
LIN {X 0,Y 587.21,Z 547.918,A -85,B 0,C 180,E1 -1288.408,E2 -1288.408} C_VEL
LIN {X 0,Y 587.195,Z 552.547,A -85,B 0,C 180,E1 -1289.388,E2 -1289.388} C_VEL
LIN {X 0,Y 587.171,Z 556.537,A -85,B 0,C 180,E1 -1290.482,E2 -1290.482} C_VEL
LIN {X 0,Y 587.136,Z 559.864,A -85,B 0,C 180,E1 -1291.802,E2 -1291.802} C_VEL
LIN {X 0,Y 587.141,Z 561.596,A -85,B 0,C 180,E1 -1293.081,E2 -1293.081} C_VEL
LIN {X 0,Y 587.133,Z 561.945,A -85,B 0,C 180,E1 -1294.316,E2 -1294.316} C_VEL
LIN {X 0,Y 587.138,Z 561.069,A -85,B 0,C 180,E1 -1295.515,E2 -1295.515} C_VEL
LIN {X 0,Y 587.134,Z 558.848,A -85,B 0,C 180,E1 -1296.763,E2 -1296.763} C_VEL
LIN {X 0,Y 587.182,Z 554.81,A -85,B 0,C 180,E1 -1298.128,E2 -1298.128} C_VEL
LIN {X 0,Y 587.203,Z 549.532,A -85,B 0,C 180,E1 -1299.371,E2 -1299.371} C_VEL
LIN {X 0,Y 587.202,Z 543.429,A -85,B 0,C 180,E1 -1300.463,E2 -1300.463} C_VEL
LIN {X 0,Y 587.243,Z 537.005,A -85,B 0,C 180,E1 -1301.394,E2 -1301.394} C_VEL
LIN {X 0,Y 587.312,Z 528.263,A -85,B 0,C 180,E1 -1302.424,E2 -1302.424} C_VEL
LIN {X 0,Y 587.389,Z 518.035,A -85,B 0,C 180,E1 -1303.391,E2 -1303.391} C_VEL
LIN {X 0,Y 587.446,Z 508.419,A -85,B 0,C 180,E1 -1304.125,E2 -1304.125} C_VEL
LIN {X 0,Y 587.516,Z 497.723,A -85,B 0,C 180,E1 -1304.787,E2 -1304.787} C_VEL
LIN {X 0,Y 587.589,Z 487.17,A -85,B 0,C 180,E1 -1305.308,E2 -1305.308} C_VEL
LIN {X 0,Y 587.649,Z 476.926,A -85,B 0,C 180,E1 -1305.705,E2 -1305.705} C_VEL
LIN {X 0,Y 587.377,Z 475.318,A -85,B 0,C 180,E1 -1305.785,E2 -1305.785} C_VEL
LIN {X 0,Y 587.315,Z 475.326,A -85,B 0,C 180,E1 -1308.928,E2 -1308.928} C_VEL
LIN {X 0,Y 587.329,Z 475.324,A -85,B 0,C 180,E1 -1311.52,E2 -1311.52} C_VEL
LIN {X 0,Y 587.283,Z 475.333,A -85,B 0,C 180,E1 -1314.099,E2 -1314.099} C_VEL
LIN {X 0,Y 587.338,Z 475.324,A -85,B 0,C 180,E1 -1316.603,E2 -1316.603} C_VEL
LIN {X 0,Y 587.325,Z 475.325,A -85,B 0,C 180,E1 -1319.493,E2 -1319.493} C_VEL
LIN {X 0,Y 587.358,Z 475.32,A -85,B 0,C 180,E1 -1322.307,E2 -1322.307} C_VEL
LIN {X 0,Y 587.335,Z 475.328,A -85,B 0,C 180,E1 -1324.483,E2 -1324.483} C_VEL
LIN {X 0,Y 587.344,Z 475.326,A -85,B 0,C 180,E1 -1327.486,E2 -1327.486} C_VEL
LIN {X 0,Y 587.325,Z 475.324,A -85,B 0,C 180,E1 -1329.695,E2 -1329.695} C_VEL
LIN {X 0,Y 587.289,Z 475.334,A -85,B 0,C 180,E1 -1331.872,E2 -1331.872} C_VEL
LIN {X 0,Y 587.326,Z 475.324,A -85,B 0,C 180,E1 -1334.025,E2 -1334.025} C_VEL
LIN {X 0,Y 587.359,Z 475.323,A -85,B 0,C 180,E1 -1336.154,E2 -1336.154} C_VEL
LIN {X 0,Y 587.344,Z 475.323,A -85,B 0,C 180,E1 -1338.962,E2 -1338.962} C_VEL
LIN {X 0,Y 587.348,Z 475.321,A -85,B 0,C 180,E1 -1341.744,E2 -1341.744} C_VEL
LIN {X 0,Y 587.343,Z 475.322,A -85,B 0,C 180,E1 -1344.507,E2 -1344.507} C_VEL
LIN {X 0,Y 587.367,Z 475.32,A -85,B 0,C 180,E1 -1347.257,E2 -1347.257} C_VEL
LIN {X 0,Y 587.387,Z 475.32,A -85,B 0,C 180,E1 -1350,E2 -1350} C_VEL
LIN {X 0,Y 587.374,Z 475.322,A -85,B 0,C 180,E1 -1352.743,E2 -1352.743} C_VEL
LIN {X 0,Y 587.342,Z 475.324,A -85,B 0,C 180,E1 -1355.493,E2 -1355.493} C_VEL
LIN {X 0,Y 587.37,Z 475.318,A -85,B 0,C 180,E1 -1358.255,E2 -1358.255} C_VEL
LIN {X 0,Y 587.337,Z 475.323,A -85,B 0,C 180,E1 -1361.124,E2 -1361.124} C_VEL
LIN {X 0,Y 587.372,Z 475.318,A -85,B 0,C 180,E1 -1364.26,E2 -1364.26} C_VEL
LIN {X 0,Y 587.31,Z 475.327,A -85,B 0,C 180,E1 -1367.407,E2 -1367.407} C_VEL
LIN {X 0,Y 587.318,Z 475.327,A -85,B 0,C 180,E1 -1369.576,E2 -1369.576} C_VEL
LIN {X 0,Y 587.321,Z 475.325,A -85,B 0,C 180,E1 -1371.774,E2 -1371.774} C_VEL
LIN {X 0,Y 587.316,Z 475.326,A -85,B 0,C 180,E1 -1374.76,E2 -1374.76} C_VEL
LIN {X 0,Y 587.321,Z 475.327,A -85,B 0,C 180,E1 -1377.047,E2 -1377.047} C_VEL
LIN {X 0,Y 587.32,Z 475.326,A -85,B 0,C 180,E1 -1379.381,E2 -1379.381} C_VEL
LIN {X 0,Y 587.349,Z 475.321,A -85,B 0,C 180,E1 -1381.835,E2 -1381.835} C_VEL
LIN {X 0,Y 587.337,Z 475.327,A -85,B 0,C 180,E1 -1384.345,E2 -1384.345} C_VEL
LIN {X 0,Y 587.349,Z 475.322,A -85,B 0,C 180,E1 -1387.607,E2 -1387.607} C_VEL
LIN {X 0,Y 587.309,Z 475.331,A -85,B 0,C 180,E1 -1390.255,E2 -1390.255} C_VEL
LIN {X 0,Y 587.318,Z 475.329,A -85,B 0,C 180,E1 -1393.118,E2 -1393.118} C_VEL
LIN {X 0,Y 587.303,Z 475.33,A -85,B 0,C 180,E1 -1396.047,E2 -1396.047} C_VEL
LIN {X 0,Y 587.337,Z 475.325,A -85,B 0,C 180,E1 -1398.925,E2 -1398.925} C_VEL
LIN {X 0,Y 587.321,Z 475.325,A -85,B 0,C 180,E1 -1401.519,E2 -1401.519} C_VEL
LIN {X 0,Y 587.301,Z 475.327,A -85,B 0,C 180,E1 -1404.462,E2 -1404.462} C_VEL
LIN {X 0,Y 587.341,Z 475.325,A -85,B 0,C 180,E1 -1406.888,E2 -1406.888} C_VEL
LIN {X 0,Y 587.335,Z 475.327,A -85,B 0,C 180,E1 -1409.83,E2 -1409.83} C_VEL
LIN {X 0,Y 587.346,Z 475.323,A -85,B 0,C 180,E1 -1412.309,E2 -1412.309} C_VEL
LIN {X 0,Y 587.356,Z 475.323,A -85,B 0,C 180,E1 -1415.42,E2 -1415.42} C_VEL
LIN {X 0,Y 587.323,Z 475.325,A -85,B 0,C 180,E1 -1418.225,E2 -1418.225} C_VEL
LIN {X 0,Y 587.337,Z 475.323,A -85,B 0,C 180,E1 -1421.15,E2 -1421.15} C_VEL
LIN {X 0,Y 587.323,Z 475.324,A -85,B 0,C 180,E1 -1424.024,E2 -1424.024} C_VEL
LIN {X 0,Y 587.355,Z 475.326,A -85,B 0,C 180,E1 -1426.154,E2 -1426.154} C_VEL
LIN {X 0,Y 587.344,Z 475.325,A -85,B 0,C 180,E1 -1428.962,E2 -1428.962} C_VEL
LIN {X 0,Y 587.341,Z 475.324,A -85,B 0,C 180,E1 -1431.744,E2 -1431.744} C_VEL
LIN {X 0,Y 587.353,Z 475.321,A -85,B 0,C 180,E1 -1434.507,E2 -1434.507} C_VEL
LIN {X 0,Y 587.356,Z 475.32,A -85,B 0,C 180,E1 -1437.256,E2 -1437.256} C_VEL
LIN {X 0,Y 587.387,Z 475.318,A -85,B 0,C 180,E1 -1440,E2 -1440} C_VEL
LIN {X 0,Y 587.37,Z 475.322,A -85,B 0,C 180,E1 -1442.743,E2 -1442.743} C_VEL
LIN {X 0,Y 587.347,Z 475.326,A -85,B 0,C 180,E1 -1445.493,E2 -1445.493} C_VEL
LIN {X 0,Y 587.368,Z 475.32,A -85,B 0,C 180,E1 -1448.255,E2 -1448.255} C_VEL
LIN {X 0,Y 587.352,Z 475.322,A -85,B 0,C 180,E1 -1451.133,E2 -1451.133} C_VEL
LIN {X 0,Y 587.363,Z 475.319,A -85,B 0,C 180,E1 -1453.846,E2 -1453.846} C_VEL
LIN {X 0,Y 587.319,Z 475.325,A -85,B 0,C 180,E1 -1456.803,E2 -1456.803} C_VEL
LIN {X 0,Y 587.317,Z 475.325,A -85,B 0,C 180,E1 -1459.576,E2 -1459.576} C_VEL
LIN {X 0,Y 587.308,Z 475.329,A -85,B 0,C 180,E1 -1461.775,E2 -1461.775} C_VEL
LIN {X 0,Y 587.353,Z 475.323,A -85,B 0,C 180,E1 -1464.758,E2 -1464.758} C_VEL
LIN {X 0,Y 587.301,Z 475.33,A -85,B 0,C 180,E1 -1467.82,E2 -1467.82} C_VEL
LIN {X 0,Y 587.339,Z 475.323,A -85,B 0,C 180,E1 -1470.51,E2 -1470.51} C_VEL
LIN {X 0,Y 587.327,Z 475.324,A -85,B 0,C 180,E1 -1473.397,E2 -1473.397} C_VEL
LIN {X 0,Y 587.298,Z 475.329,A -85,B 0,C 180,E1 -1475.9,E2 -1475.9} C_VEL
LIN {X 0,Y 587.321,Z 475.33,A -85,B 0,C 180,E1 -1478.48,E2 -1478.48} C_VEL
LIN {X 0,Y 587.334,Z 475.325,A -85,B 0,C 180,E1 -1481.157,E2 -1481.157} C_VEL
LIN {X 0,Y 587.314,Z 475.327,A -85,B 0,C 180,E1 -1484.112,E2 -1484.112} C_VEL
LIN {X 0,Y 587.304,Z 475.327,A -85,B 0,C 180,E1 -1486.992,E2 -1486.992} C_VEL
LIN {X 0,Y 587.338,Z 475.327,A -85,B 0,C 180,E1 -1488.925,E2 -1488.925} C_VEL
LIN {X 0,Y 587.316,Z 475.327,A -85,B 0,C 180,E1 -1491.519,E2 -1491.519} C_VEL
LIN {X 0,Y 587.33,Z 475.382,A -85,B 0,C 180,E1 -1493.572,E2 -1493.572} C_VEL
LIN {X 0,Y 587.935,Z 479.118,A -85,B 0,C 180,E1 -1494.376,E2 -1494.376} C_VEL
LIN {X 0,Y 587.881,Z 491.16,A -85,B 0,C 180,E1 -1496.808,E2 -1496.808} C_VEL
LIN {X 0,Y 587.947,Z 504.597,A -85,B 0,C 180,E1 -1499.39,E2 -1499.39} C_VEL
LIN {X 0,Y 587.867,Z 516.93,A -85,B 0,C 180,E1 -1501.821,E2 -1501.821} C_VEL
LIN {X 0,Y 587.736,Z 530.625,A -85,B 0,C 180,E1 -1504.502,E2 -1504.502} C_VEL
LIN {X 0,Y 587.652,Z 545.108,A -85,B 0,C 180,E1 -1507.277,E2 -1507.277} C_VEL
LIN {X 0,Y 587.505,Z 561.927,A -85,B 0,C 180,E1 -1510.431,E2 -1510.431} C_VEL
LIN {X 0,Y 587.422,Z 577.579,A -85,B 0,C 180,E1 -1513.313,E2 -1513.313} C_VEL
LIN {X 0,Y 587.322,Z 595.187,A -85,B 0,C 180,E1 -1516.506,E2 -1516.506} C_VEL
LIN {X 0,Y 587.315,Z 602.157,A -85,B 0,C 180,E1 -1517.759,E2 -1517.759} C_VEL
LIN {X 0,Y 587.745,Z 607.948,A -85,B 0,C 180,E1 -1517.855,E2 -1517.855} C_VEL
LIN {X 0,Y 587.673,Z 621.219,A -85,B 0,C 180,E1 -1518.16,E2 -1518.16} C_VEL
LIN {X 0,Y 587.631,Z 633.746,A -85,B 0,C 180,E1 -1518.59,E2 -1518.59} C_VEL
LIN {X 0,Y 587.522,Z 645.633,A -85,B 0,C 180,E1 -1519.14,E2 -1519.14} C_VEL
LIN {X 0,Y 587.468,Z 657.201,A -85,B 0,C 180,E1 -1519.837,E2 -1519.837} C_VEL
LIN {X 0,Y 587.366,Z 667.597,A -85,B 0,C 180,E1 -1520.617,E2 -1520.617} C_VEL
LIN {X 0,Y 587.321,Z 676.112,A -85,B 0,C 180,E1 -1521.398,E2 -1521.398} C_VEL
LIN {X 0,Y 587.274,Z 683.961,A -85,B 0,C 180,E1 -1522.263,E2 -1522.263} C_VEL
LIN {X 0,Y 587.23,Z 690.47,A -85,B 0,C 180,E1 -1523.126,E2 -1523.126} C_VEL
LIN {X 0,Y 587.236,Z 696.867,A -85,B 0,C 180,E1 -1524.161,E2 -1524.161} C_VEL
LIN {X 0,Y 587.147,Z 701.95,A -85,B 0,C 180,E1 -1525.194,E2 -1525.194} C_VEL
LIN {X 0,Y 587.213,Z 705.896,A -85,B 0,C 180,E1 -1526.226,E2 -1526.226} C_VEL
LIN {X 0,Y 587.132,Z 708.809,A -85,B 0,C 180,E1 -1527.256,E2 -1527.256} C_VEL
LIN {X 0,Y 587.14,Z 710.201,A -85,B 0,C 180,E1 -1527.942,E2 -1527.942} C_VEL
LIN {X 0,Y 587.14,Z 711.784,A -85,B 0,C 180,E1 -1529.314,E2 -1529.314} C_VEL
LIN {X 0,Y 587.137,Z 712,A -85,B 0,C 180,E1 -1530,E2 -1530} C_VEL
LIN {X 0,Y 587.147,Z 711.185,A -85,B 0,C 180,E1 -1531.372,E2 -1531.372} C_VEL
LIN {X 0,Y 587.14,Z 710.201,A -85,B 0,C 180,E1 -1532.058,E2 -1532.058} C_VEL
LIN {X 0,Y 587.132,Z 708.809,A -85,B 0,C 180,E1 -1532.744,E2 -1532.744} C_VEL
LIN {X 0,Y 587.213,Z 705.896,A -85,B 0,C 180,E1 -1533.774,E2 -1533.774} C_VEL
LIN {X 0,Y 587.147,Z 701.949,A -85,B 0,C 180,E1 -1534.806,E2 -1534.806} C_VEL
LIN {X 0,Y 587.217,Z 695.877,A -85,B 0,C 180,E1 -1536.011,E2 -1536.011} C_VEL
LIN {X 0,Y 587.245,Z 689.235,A -85,B 0,C 180,E1 -1537.046,E2 -1537.046} C_VEL
LIN {X 0,Y 587.3,Z 680.989,A -85,B 0,C 180,E1 -1538.083,E2 -1538.083} C_VEL
LIN {X 0,Y 587.343,Z 672.536,A -85,B 0,C 180,E1 -1538.949,E2 -1538.949} C_VEL
LIN {X 0,Y 587.42,Z 662.092,A -85,B 0,C 180,E1 -1539.816,E2 -1539.816} C_VEL
LIN {X 0,Y 587.497,Z 651.756,A -85,B 0,C 180,E1 -1540.511,E2 -1540.511} C_VEL
LIN {X 0,Y 587.56,Z 640.066,A -85,B 0,C 180,E1 -1541.137,E2 -1541.137} C_VEL
LIN {X 0,Y 587.624,Z 627.64,A -85,B 0,C 180,E1 -1541.638,E2 -1541.638} C_VEL
LIN {X 0,Y 587.713,Z 614.43,A -85,B 0,C 180,E1 -1542.014,E2 -1542.014} C_VEL
LIN {X 0,Y 587.52,Z 603.59,A -85,B 0,C 180,E1 -1542.215,E2 -1542.215} C_VEL
LIN {X 0,Y 587.32,Z 602.033,A -85,B 0,C 180,E1 -1542.263,E2 -1542.263} C_VEL
LIN {X 0,Y 587.338,Z 587.36,A -85,B 0,C 180,E1 -1544.908,E2 -1544.908} C_VEL
LIN {X 0,Y 587.458,Z 571.709,A -85,B 0,C 180,E1 -1547.762,E2 -1547.762} C_VEL
LIN {X 0,Y 587.519,Z 556.057,A -85,B 0,C 180,E1 -1550.664,E2 -1550.664} C_VEL
LIN {X 0,Y 587.645,Z 542.362,A -85,B 0,C 180,E1 -1553.245,E2 -1553.245} C_VEL
LIN {X 0,Y 587.757,Z 528.667,A -85,B 0,C 180,E1 -1555.877,E2 -1555.877} C_VEL
LIN {X 0,Y 587.875,Z 514.972,A -85,B 0,C 180,E1 -1558.568,E2 -1558.568} C_VEL
LIN {X 0,Y 587.947,Z 504.542,A -85,B 0,C 180,E1 -1560.61,E2 -1560.61} C_VEL
LIN {X 0,Y 587.806,Z 489.702,A -85,B 0,C 180,E1 -1563.367,E2 -1563.367} C_VEL
LIN {X 0,Y 587.75,Z 478.171,A -85,B 0,C 180,E1 -1565.599,E2 -1565.599} C_VEL
LIN {X 0,Y 587.324,Z 475.33,A -85,B 0,C 180,E1 -1566.216,E2 -1566.216} C_VEL
LIN {X 0,Y 587.323,Z 475.328,A -85,B 0,C 180,E1 -1568.94,E2 -1568.94} C_VEL
LIN {X 0,Y 587.357,Z 475.323,A -85,B 0,C 180,E1 -1572.073,E2 -1572.073} C_VEL
LIN {X 0,Y 587.321,Z 475.329,A -85,B 0,C 180,E1 -1575.089,E2 -1575.089} C_VEL
LIN {X 0,Y 587.357,Z 475.322,A -85,B 0,C 180,E1 -1577.928,E2 -1577.928} C_VEL
LIN {X 0,Y 587.326,Z 475.329,A -85,B 0,C 180,E1 -1581.06,E2 -1581.06} C_VEL
LIN {X 0,Y 587.321,Z 475.327,A -85,B 0,C 180,E1 -1583.297,E2 -1583.297} C_VEL
LIN {X 0,Y 587.335,Z 475.325,A -85,B 0,C 180,E1 -1585.778,E2 -1585.778} C_VEL
LIN {X 0,Y 587.345,Z 475.323,A -85,B 0,C 180,E1 -1588.231,E2 -1588.231} C_VEL
LIN {X 0,Y 587.353,Z 475.323,A -85,B 0,C 180,E1 -1590.867,E2 -1590.867} C_VEL
LIN {X 0,Y 587.343,Z 475.325,A -85,B 0,C 180,E1 -1593.823,E2 -1593.823} C_VEL
LIN {X 0,Y 587.332,Z 475.328,A -85,B 0,C 180,E1 -1595.993,E2 -1595.993} C_VEL
LIN {X 0,Y 587.328,Z 475.326,A -85,B 0,C 180,E1 -1598.226,E2 -1598.226} C_VEL
LIN {X 0,Y 587.351,Z 475.325,A -85,B 0,C 180,E1 -1601.151,E2 -1601.151} C_VEL
LIN {X 0,Y 587.328,Z 475.326,A -85,B 0,C 180,E1 -1604.025,E2 -1604.025} C_VEL
LIN {X 0,Y 587.315,Z 475.327,A -85,B 0,C 180,E1 -1606.858,E2 -1606.858} C_VEL
LIN {X 0,Y 587.338,Z 475.327,A -85,B 0,C 180,E1 -1609.66,E2 -1609.66} C_VEL
LIN {X 0,Y 587.355,Z 475.324,A -85,B 0,C 180,E1 -1612.437,E2 -1612.437} C_VEL
LIN {X 0,Y 587.353,Z 475.322,A -85,B 0,C 180,E1 -1615.195,E2 -1615.195} C_VEL
LIN {X 0,Y 587.376,Z 475.319,A -85,B 0,C 180,E1 -1617.943,E2 -1617.943} C_VEL
LIN {X 0,Y 587.391,Z 475.319,A -85,B 0,C 180,E1 -1620.686,E2 -1620.686} C_VEL
LIN {X 0,Y 587.332,Z 475.329,A -85,B 0,C 180,E1 -1623.43,E2 -1623.43} C_VEL
LIN {X 0,Y 587.346,Z 475.323,A -85,B 0,C 180,E1 -1625.493,E2 -1625.493} C_VEL
LIN {X 0,Y 587.369,Z 475.323,A -85,B 0,C 180,E1 -1628.255,E2 -1628.255} C_VEL
LIN {X 0,Y 587.355,Z 475.324,A -85,B 0,C 180,E1 -1631.134,E2 -1631.134} C_VEL
LIN {X 0,Y 587.371,Z 475.321,A -85,B 0,C 180,E1 -1634.261,E2 -1634.261} C_VEL
LIN {X 0,Y 587.349,Z 475.325,A -85,B 0,C 180,E1 -1637.406,E2 -1637.406} C_VEL
LIN {X 0,Y 587.313,Z 475.328,A -85,B 0,C 180,E1 -1638.292,E2 -1638.292} C_VEL
LIN {X 0,Y 586.668,Z 475.409,A -85,B 0,C 180,E1 -1638.864,E2 -1638.864} C_VEL
LIN {X 0,Y 583.848,Z 475.762,A -85,B 0,C 180,E1 -1639.792,E2 -1639.792} C_VEL
LIN {X 0,Y 581.441,Z 476.062,A -85,B 0,C 180,E1 -1640.539,E2 -1640.539} C_VEL
LIN {X 0,Y 580.386,Z 476.193,A -85,B 0,C 180,E1 -1641.116,E2 -1641.116} C_VEL
LIN {X 0,Y 580.289,Z 476.203,A -85,B 0,C 180,E1 -1641.311,E2 -1641.311} C_VEL
LIN {X 0,Y 580.303,Z 476.33,A -85,B 0,C 180,E1 -1642.216,E2 -1642.216} C_VEL
LIN {X 0,Y 580.653,Z 479.09,A -85,B 0,C 180,E1 -1642.319,E2 -1642.319} C_VEL
LIN {X 0,Y 580.592,Z 490.417,A -85,B 0,C 180,E1 -1642.79,E2 -1642.79} C_VEL
LIN {X 0,Y 580.497,Z 502.826,A -85,B 0,C 180,E1 -1643.471,E2 -1643.471} C_VEL
LIN {X 0,Y 580.378,Z 513.513,A -85,B 0,C 180,E1 -1644.218,E2 -1644.218} C_VEL
LIN {X 0,Y 580.284,Z 523.488,A -85,B 0,C 180,E1 -1645.081,E2 -1645.081} C_VEL
LIN {X 0,Y 580.213,Z 532.87,A -85,B 0,C 180,E1 -1646.084,E2 -1646.084} C_VEL
LIN {X 0,Y 580.149,Z 541.302,A -85,B 0,C 180,E1 -1647.214,E2 -1647.214} C_VEL
LIN {X 0,Y 580.131,Z 547.163,A -85,B 0,C 180,E1 -1648.195,E2 -1648.195} C_VEL
LIN {X 0,Y 580.101,Z 552.305,A -85,B 0,C 180,E1 -1649.274,E2 -1649.274} C_VEL
LIN {X 0,Y 580.08,Z 555.747,A -85,B 0,C 180,E1 -1650.186,E2 -1650.186} C_VEL
LIN {X 0,Y 580.033,Z 559.076,A -85,B 0,C 180,E1 -1651.401,E2 -1651.401} C_VEL
LIN {X 0,Y 580.04,Z 560.61,A -85,B 0,C 180,E1 -1652.217,E2 -1652.217} C_VEL
LIN {X 0,Y 580.061,Z 561.737,A -85,B 0,C 180,E1 -1653.279,E2 -1653.279} C_VEL
LIN {X 0,Y 580.019,Z 561.877,A -85,B 0,C 180,E1 -1654.518,E2 -1654.518} C_VEL
LIN {X 0,Y 580.03,Z 560.81,A -85,B 0,C 180,E1 -1655.726,E2 -1655.726} C_VEL
LIN {X 0,Y 580.049,Z 558.611,A -85,B 0,C 180,E1 -1656.901,E2 -1656.901} C_VEL
LIN {X 0,Y 580.098,Z 554.87,A -85,B 0,C 180,E1 -1658.162,E2 -1658.162} C_VEL
LIN {X 0,Y 580.09,Z 550.832,A -85,B 0,C 180,E1 -1659.16,E2 -1659.16} C_VEL
LIN {X 0,Y 580.154,Z 545.167,A -85,B 0,C 180,E1 -1660.254,E2 -1660.254} C_VEL
LIN {X 0,Y 580.171,Z 538.233,A -85,B 0,C 180,E1 -1661.318,E2 -1661.318} C_VEL
LIN {X 0,Y 580.247,Z 530.968,A -85,B 0,C 180,E1 -1662.226,E2 -1662.226} C_VEL
LIN {X 0,Y 580.298,Z 522.944,A -85,B 0,C 180,E1 -1663.06,E2 -1663.06} C_VEL
LIN {X 0,Y 580.427,Z 513.344,A -85,B 0,C 180,E1 -1663.885,E2 -1663.885} C_VEL
LIN {X 0,Y 580.473,Z 503.024,A -85,B 0,C 180,E1 -1664.607,E2 -1664.607} C_VEL
LIN {X 0,Y 580.567,Z 491.505,A -85,B 0,C 180,E1 -1665.248,E2 -1665.248} C_VEL
LIN {X 0,Y 580.681,Z 479.004,A -85,B 0,C 180,E1 -1665.774,E2 -1665.774} C_VEL
LIN {X 0,Y 580.326,Z 476.197,A -85,B 0,C 180,E1 -1665.892,E2 -1665.892} C_VEL
LIN {X 0,Y 580.285,Z 476.203,A -85,B 0,C 180,E1 -1669.155,E2 -1669.155} C_VEL
LIN {X 0,Y 580.293,Z 476.201,A -85,B 0,C 180,E1 -1671.927,E2 -1671.927} C_VEL
LIN {X 0,Y 580.235,Z 476.208,A -85,B 0,C 180,E1 -1674.451,E2 -1674.451} C_VEL
LIN {X 0,Y 580.294,Z 476.206,A -85,B 0,C 180,E1 -1676.975,E2 -1676.975} C_VEL
LIN {X 0,Y 580.286,Z 476.202,A -85,B 0,C 180,E1 -1679.424,E2 -1679.424} C_VEL
LIN {X 0,Y 580.304,Z 476.198,A -85,B 0,C 180,E1 -1682.141,E2 -1682.141} C_VEL
LIN {X 0,Y 580.293,Z 476.201,A -85,B 0,C 180,E1 -1684.919,E2 -1684.919} C_VEL
LIN {X 0,Y 580.277,Z 476.202,A -85,B 0,C 180,E1 -1687.947,E2 -1687.947} C_VEL
LIN {X 0,Y 580.288,Z 476.201,A -85,B 0,C 180,E1 -1690.913,E2 -1690.913} C_VEL
LIN {X 0,Y 580.276,Z 476.203,A -85,B 0,C 180,E1 -1693.825,E2 -1693.825} C_VEL
LIN {X 0,Y 580.319,Z 476.198,A -85,B 0,C 180,E1 -1695.983,E2 -1695.983} C_VEL
LIN {X 0,Y 580.312,Z 476.198,A -85,B 0,C 180,E1 -1698.827,E2 -1698.827} C_VEL
LIN {X 0,Y 580.317,Z 476.197,A -85,B 0,C 180,E1 -1701.644,E2 -1701.644} C_VEL
LIN {X 0,Y 580.31,Z 476.198,A -85,B 0,C 180,E1 -1704.44,E2 -1704.44} C_VEL
LIN {X 0,Y 580.335,Z 476.196,A -85,B 0,C 180,E1 -1707.223,E2 -1707.223} C_VEL
LIN {X 0,Y 580.357,Z 476.196,A -85,B 0,C 180,E1 -1710,E2 -1710} C_VEL
LIN {X 0,Y 580.34,Z 476.199,A -85,B 0,C 180,E1 -1712.776,E2 -1712.776} C_VEL
LIN {X 0,Y 580.31,Z 476.201,A -85,B 0,C 180,E1 -1715.56,E2 -1715.56} C_VEL
LIN {X 0,Y 580.333,Z 476.196,A -85,B 0,C 180,E1 -1718.356,E2 -1718.356} C_VEL
LIN {X 0,Y 580.307,Z 476.199,A -85,B 0,C 180,E1 -1721.191,E2 -1721.191} C_VEL
LIN {X 0,Y 580.333,Z 476.195,A -85,B 0,C 180,E1 -1724.017,E2 -1724.017} C_VEL
LIN {X 0,Y 580.296,Z 476.2,A -85,B 0,C 180,E1 -1726.906,E2 -1726.906} C_VEL
LIN {X 0,Y 580.293,Z 476.2,A -85,B 0,C 180,E1 -1729.823,E2 -1729.823} C_VEL
LIN {X 0,Y 580.273,Z 476.206,A -85,B 0,C 180,E1 -1732.053,E2 -1732.053} C_VEL
LIN {X 0,Y 580.291,Z 476.203,A -85,B 0,C 180,E1 -1735.081,E2 -1735.081} C_VEL
LIN {X 0,Y 580.261,Z 476.205,A -85,B 0,C 180,E1 -1737.85,E2 -1737.85} C_VEL
LIN {X 0,Y 580.278,Z 476.202,A -85,B 0,C 180,E1 -1740.692,E2 -1740.692} C_VEL
LIN {X 0,Y 580.287,Z 476.201,A -85,B 0,C 180,E1 -1743.313,E2 -1743.313} C_VEL
LIN {X 0,Y 580.236,Z 476.212,A -85,B 0,C 180,E1 -1745.754,E2 -1745.754} C_VEL
LIN {X 0,Y 580.292,Z 476.2,A -85,B 0,C 180,E1 -1748.146,E2 -1748.146} C_VEL
LIN {X 0,Y 580.283,Z 476.202,A -85,B 0,C 180,E1 -1750.845,E2 -1750.845} C_VEL
LIN {X 0,Y 580.284,Z 476.202,A -85,B 0,C 180,E1 -1753.658,E2 -1753.658} C_VEL
LIN {X 0,Y 580.24,Z 476.208,A -85,B 0,C 180,E1 -1756.613,E2 -1756.613} C_VEL
LIN {X 0,Y 580.3,Z 476.204,A -85,B 0,C 180,E1 -1759.156,E2 -1759.156} C_VEL
LIN {X 0,Y 580.285,Z 476.204,A -85,B 0,C 180,E1 -1761.928,E2 -1761.928} C_VEL
LIN {X 0,Y 580.256,Z 476.205,A -85,B 0,C 180,E1 -1764.452,E2 -1764.452} C_VEL
LIN {X 0,Y 580.292,Z 476.203,A -85,B 0,C 180,E1 -1766.975,E2 -1766.975} C_VEL
LIN {X 0,Y 580.295,Z 476.203,A -85,B 0,C 180,E1 -1769.425,E2 -1769.425} C_VEL
LIN {X 0,Y 580.296,Z 476.2,A -85,B 0,C 180,E1 -1772.142,E2 -1772.142} C_VEL
LIN {X 0,Y 580.323,Z 476.198,A -85,B 0,C 180,E1 -1775.27,E2 -1775.27} C_VEL
LIN {X 0,Y 580.274,Z 476.202,A -85,B 0,C 180,E1 -1777.947,E2 -1777.947} C_VEL
LIN {X 0,Y 580.289,Z 476.201,A -85,B 0,C 180,E1 -1780.913,E2 -1780.913} C_VEL
LIN {X 0,Y 580.274,Z 476.202,A -85,B 0,C 180,E1 -1783.825,E2 -1783.825} C_VEL
LIN {X 0,Y 580.315,Z 476.201,A -85,B 0,C 180,E1 -1785.983,E2 -1785.983} C_VEL
LIN {X 0,Y 580.309,Z 476.2,A -85,B 0,C 180,E1 -1788.827,E2 -1788.827} C_VEL
LIN {X 0,Y 580.31,Z 476.199,A -85,B 0,C 180,E1 -1791.643,E2 -1791.643} C_VEL
LIN {X 0,Y 580.319,Z 476.197,A -85,B 0,C 180,E1 -1794.44,E2 -1794.44} C_VEL
LIN {X 0,Y 580.325,Z 476.196,A -85,B 0,C 180,E1 -1797.223,E2 -1797.223} C_VEL
LIN {X 0,Y 580.356,Z 476.193,A -85,B 0,C 180,E1 -1800,E2 -1800} C_VEL
LIN {X 0,Y 580.334,Z 476.198,A -85,B 0,C 180,E1 -1802.776,E2 -1802.776} C_VEL
LIN {X 0,Y 580.314,Z 476.203,A -85,B 0,C 180,E1 -1805.56,E2 -1805.56} C_VEL
LIN {X 0,Y 580.329,Z 476.198,A -85,B 0,C 180,E1 -1808.356,E2 -1808.356} C_VEL
LIN {X 0,Y 580.304,Z 476.2,A -85,B 0,C 180,E1 -1811.191,E2 -1811.191} C_VEL
LIN {X 0,Y 580.32,Z 476.197,A -85,B 0,C 180,E1 -1814.017,E2 -1814.017} C_VEL
LIN {X 0,Y 580.293,Z 476.2,A -85,B 0,C 180,E1 -1816.906,E2 -1816.906} C_VEL
LIN {X 0,Y 580.291,Z 476.2,A -85,B 0,C 180,E1 -1819.823,E2 -1819.823} C_VEL
LIN {X 0,Y 580.252,Z 476.21,A -85,B 0,C 180,E1 -1822.053,E2 -1822.053} C_VEL
LIN {X 0,Y 580.308,Z 476.203,A -85,B 0,C 180,E1 -1825.08,E2 -1825.08} C_VEL
LIN {X 0,Y 580.275,Z 476.206,A -85,B 0,C 180,E1 -1828.187,E2 -1828.187} C_VEL
LIN {X 0,Y 580.287,Z 476.203,A -85,B 0,C 180,E1 -1830.694,E2 -1830.694} C_VEL
LIN {X 0,Y 580.284,Z 476.201,A -85,B 0,C 180,E1 -1833.313,E2 -1833.313} C_VEL
LIN {X 0,Y 580.251,Z 476.208,A -85,B 0,C 180,E1 -1835.757,E2 -1835.757} C_VEL
LIN {X 0,Y 580.287,Z 476.202,A -85,B 0,C 180,E1 -1838.147,E2 -1838.147} C_VEL
LIN {X 0,Y 580.294,Z 476.2,A -85,B 0,C 180,E1 -1840.844,E2 -1840.844} C_VEL
LIN {X 0,Y 580.275,Z 476.202,A -85,B 0,C 180,E1 -1843.658,E2 -1843.658} C_VEL
LIN {X 0,Y 580.244,Z 476.205,A -85,B 0,C 180,E1 -1846.613,E2 -1846.613} C_VEL
LIN {X 0,Y 580.3,Z 476.202,A -85,B 0,C 180,E1 -1849.157,E2 -1849.157} C_VEL
LIN {X 0,Y 580.282,Z 476.207,A -85,B 0,C 180,E1 -1851.928,E2 -1851.928} C_VEL
LIN {X 0,Y 580.303,Z 476.362,A -85,B 0,C 180,E1 -1853.362,E2 -1853.362} C_VEL
LIN {X 0,Y 581.018,Z 479.882,A -85,B 0,C 180,E1 -1854.138,E2 -1854.138} C_VEL
LIN {X 0,Y 581.023,Z 491.767,A -85,B 0,C 180,E1 -1856.576,E2 -1856.576} C_VEL
LIN {X 0,Y 580.984,Z 505.098,A -85,B 0,C 180,E1 -1859.19,E2 -1859.19} C_VEL
LIN {X 0,Y 580.975,Z 516.93,A -85,B 0,C 180,E1 -1861.456,E2 -1861.456} C_VEL
LIN {X 0,Y 580.812,Z 530.625,A -85,B 0,C 180,E1 -1864.176,E2 -1864.176} C_VEL
LIN {X 0,Y 580.705,Z 544.622,A -85,B 0,C 180,E1 -1866.896,E2 -1866.896} C_VEL
LIN {X 0,Y 580.518,Z 561.928,A -85,B 0,C 180,E1 -1870.185,E2 -1870.185} C_VEL
LIN {X 0,Y 580.419,Z 577.292,A -85,B 0,C 180,E1 -1873.053,E2 -1873.053} C_VEL
LIN {X 0,Y 580.3,Z 593.23,A -85,B 0,C 180,E1 -1875.982,E2 -1875.982} C_VEL
LIN {X 0,Y 580.268,Z 602.157,A -85,B 0,C 180,E1 -1877.608,E2 -1877.608} C_VEL
LIN {X 0,Y 580.804,Z 607.947,A -85,B 0,C 180,E1 -1877.708,E2 -1877.708} C_VEL
LIN {X 0,Y 580.746,Z 621.219,A -85,B 0,C 180,E1 -1878.017,E2 -1878.017} C_VEL
LIN {X 0,Y 580.675,Z 633.372,A -85,B 0,C 180,E1 -1878.437,E2 -1878.437} C_VEL
LIN {X 0,Y 580.543,Z 645.631,A -85,B 0,C 180,E1 -1879.008,E2 -1879.008} C_VEL
LIN {X 0,Y 580.445,Z 657.202,A -85,B 0,C 180,E1 -1879.712,E2 -1879.712} C_VEL
LIN {X 0,Y 580.346,Z 667.598,A -85,B 0,C 180,E1 -1880.503,E2 -1880.503} C_VEL
LIN {X 0,Y 580.271,Z 676.113,A -85,B 0,C 180,E1 -1881.292,E2 -1881.292} C_VEL
LIN {X 0,Y 580.222,Z 683.961,A -85,B 0,C 180,E1 -1882.168,E2 -1882.168} C_VEL
LIN {X 0,Y 580.153,Z 691.65,A -85,B 0,C 180,E1 -1883.222,E2 -1883.222} C_VEL
LIN {X 0,Y 580.139,Z 698.68,A -85,B 0,C 180,E1 -1884.439,E2 -1884.439} C_VEL
LIN {X 0,Y 580.108,Z 703.372,A -85,B 0,C 180,E1 -1885.483,E2 -1885.483} C_VEL
LIN {X 0,Y 580.123,Z 706.957,A -85,B 0,C 180,E1 -1886.527,E2 -1886.527} C_VEL
LIN {X 0,Y 580.043,Z 708.809,A -85,B 0,C 180,E1 -1887.222,E2 -1887.222} C_VEL
LIN {X 0,Y 580.039,Z 710.2,A -85,B 0,C 180,E1 -1887.917,E2 -1887.917} C_VEL
LIN {X 0,Y 580.04,Z 711.784,A -85,B 0,C 180,E1 -1889.306,E2 -1889.306} C_VEL
LIN {X 0,Y 580.037,Z 712,A -85,B 0,C 180,E1 -1890,E2 -1890} C_VEL
LIN {X 0,Y 580.046,Z 711.185,A -85,B 0,C 180,E1 -1891.389,E2 -1891.389} C_VEL
LIN {X 0,Y 580.039,Z 710.201,A -85,B 0,C 180,E1 -1892.083,E2 -1892.083} C_VEL
LIN {X 0,Y 580.043,Z 708.809,A -85,B 0,C 180,E1 -1892.778,E2 -1892.778} C_VEL
LIN {X 0,Y 580.11,Z 705.896,A -85,B 0,C 180,E1 -1893.821,E2 -1893.821} C_VEL
LIN {X 0,Y 580.053,Z 701.949,A -85,B 0,C 180,E1 -1894.865,E2 -1894.865} C_VEL
LIN {X 0,Y 580.139,Z 695.877,A -85,B 0,C 180,E1 -1896.085,E2 -1896.085} C_VEL
LIN {X 0,Y 580.184,Z 689.236,A -85,B 0,C 180,E1 -1897.133,E2 -1897.133} C_VEL
LIN {X 0,Y 580.251,Z 680.989,A -85,B 0,C 180,E1 -1898.182,E2 -1898.182} C_VEL
LIN {X 0,Y 580.308,Z 672.536,A -85,B 0,C 180,E1 -1899.059,E2 -1899.059} C_VEL
LIN {X 0,Y 580.424,Z 662.093,A -85,B 0,C 180,E1 -1899.936,E2 -1899.936} C_VEL
LIN {X 0,Y 580.5,Z 651.755,A -85,B 0,C 180,E1 -1900.64,E2 -1900.64} C_VEL
LIN {X 0,Y 580.573,Z 640.49,A -85,B 0,C 180,E1 -1901.252,E2 -1901.252} C_VEL
LIN {X 0,Y 580.688,Z 628.762,A -85,B 0,C 180,E1 -1901.741,E2 -1901.741} C_VEL
LIN {X 0,Y 580.756,Z 615.343,A -85,B 0,C 180,E1 -1902.138,E2 -1902.138} C_VEL
LIN {X 0,Y 580.631,Z 604.532,A -85,B 0,C 180,E1 -1902.348,E2 -1902.348} C_VEL
LIN {X 0,Y 580.252,Z 602.033,A -85,B 0,C 180,E1 -1902.415,E2 -1902.415} C_VEL
LIN {X 0,Y 580.319,Z 587.36,A -85,B 0,C 180,E1 -1905.093,E2 -1905.093} C_VEL
LIN {X 0,Y 580.441,Z 571.709,A -85,B 0,C 180,E1 -1907.984,E2 -1907.984} C_VEL
LIN {X 0,Y 580.544,Z 556.23,A -85,B 0,C 180,E1 -1910.891,E2 -1910.891} C_VEL
LIN {X 0,Y 580.674,Z 542.362,A -85,B 0,C 180,E1 -1913.541,E2 -1913.541} C_VEL
LIN {X 0,Y 580.836,Z 529.034,A -85,B 0,C 180,E1 -1916.137,E2 -1916.137} C_VEL
LIN {X 0,Y 581.001,Z 514.934,A -85,B 0,C 180,E1 -1918.938,E2 -1918.938} C_VEL
LIN {X 0,Y 580.897,Z 501.965,A -85,B 0,C 180,E1 -1921.348,E2 -1921.348} C_VEL
LIN {X 0,Y 580.832,Z 486.771,A -85,B 0,C 180,E1 -1924.226,E2 -1924.226} C_VEL
LIN {X 0,Y 580.75,Z 478.737,A -85,B 0,C 180,E1 -1925.825,E2 -1925.825} C_VEL
LIN {X 0,Y 580.267,Z 476.208,A -85,B 0,C 180,E1 -1926.404,E2 -1926.404} C_VEL
LIN {X 0,Y 580.296,Z 476.202,A -85,B 0,C 180,E1 -1929.185,E2 -1929.185} C_VEL
LIN {X 0,Y 580.302,Z 476.201,A -85,B 0,C 180,E1 -1931.767,E2 -1931.767} C_VEL
LIN {X 0,Y 580.271,Z 476.206,A -85,B 0,C 180,E1 -1934.626,E2 -1934.626} C_VEL
LIN {X 0,Y 580.289,Z 476.205,A -85,B 0,C 180,E1 -1937.628,E2 -1937.628} C_VEL
LIN {X 0,Y 580.285,Z 476.205,A -85,B 0,C 180,E1 -1940.066,E2 -1940.066} C_VEL
LIN {X 0,Y 580.291,Z 476.203,A -85,B 0,C 180,E1 -1942.731,E2 -1942.731} C_VEL
LIN {X 0,Y 580.294,Z 476.201,A -85,B 0,C 180,E1 -1945.443,E2 -1945.443} C_VEL
LIN {X 0,Y 580.307,Z 476.2,A -85,B 0,C 180,E1 -1947.969,E2 -1947.969} C_VEL
LIN {X 0,Y 580.305,Z 476.2,A -85,B 0,C 180,E1 -1950.691,E2 -1950.691} C_VEL
LIN {X 0,Y 580.293,Z 476.205,A -85,B 0,C 180,E1 -1953.667,E2 -1953.667} C_VEL
LIN {X 0,Y 580.302,Z 476.201,A -85,B 0,C 180,E1 -1955.684,E2 -1955.684} C_VEL
LIN {X 0,Y 580.29,Z 476.204,A -85,B 0,C 180,E1 -1958.695,E2 -1958.695} C_VEL
LIN {X 0,Y 580.3,Z 476.203,A -85,B 0,C 180,E1 -1960.914,E2 -1960.914} C_VEL
LIN {X 0,Y 580.277,Z 476.205,A -85,B 0,C 180,E1 -1963.826,E2 -1963.826} C_VEL
LIN {X 0,Y 580.272,Z 476.204,A -85,B 0,C 180,E1 -1966.696,E2 -1966.696} C_VEL
LIN {X 0,Y 580.298,Z 476.202,A -85,B 0,C 180,E1 -1969.533,E2 -1969.533} C_VEL
LIN {X 0,Y 580.322,Z 476.201,A -85,B 0,C 180,E1 -1972.345,E2 -1972.345} C_VEL
LIN {X 0,Y 580.327,Z 476.197,A -85,B 0,C 180,E1 -1975.137,E2 -1975.137} C_VEL
LIN {X 0,Y 580.346,Z 476.195,A -85,B 0,C 180,E1 -1977.918,E2 -1977.918} C_VEL
LIN {X 0,Y 580.363,Z 476.194,A -85,B 0,C 180,E1 -1980.694,E2 -1980.694} C_VEL
LIN {X 0,Y 580.284,Z 476.207,A -85,B 0,C 180,E1 -1983.472,E2 -1983.472} C_VEL
LIN {X 0,Y 580.313,Z 476.2,A -85,B 0,C 180,E1 -1985.56,E2 -1985.56} C_VEL
LIN {X 0,Y 580.331,Z 476.2,A -85,B 0,C 180,E1 -1988.356,E2 -1988.356} C_VEL
LIN {X 0,Y 580.306,Z 476.201,A -85,B 0,C 180,E1 -1991.191,E2 -1991.191} C_VEL
LIN {X 0,Y 580.331,Z 476.197,A -85,B 0,C 180,E1 -1994.017,E2 -1994.017} C_VEL
LIN {X 0,Y 580.319,Z 476.201,A -85,B 0,C 180,E1 -1996.914,E2 -1996.914} C_VEL
LIN {X 0,Y 580.291,Z 476.205,A -85,B 0,C 180,E1 -1999.823,E2 -1999.823} C_VEL
LIN {X 0,Y 580.289,Z 476.203,A -85,B 0,C 180,E1 -2001.311,E2 -2001.311} C_VEL
LIN {X 0,Y 579.998,Z 476.852,A -85,B 0,C 180,E1 -2001.623,E2 -2001.623} C_VEL
LIN {X 0,Y 579.117,Z 479.005,A -85,B 0,C 180,E1 -2001.971,E2 -2001.971} C_VEL
LIN {X 0,Y 577.5,Z 483.263,A -85,B 0,C 180,E1 -2002.342,E2 -2002.342} C_VEL
LIN {X 0,Y 575.707,Z 489.08,A -85,B 0,C 180,E1 -2002.634,E2 -2002.634} C_VEL
LIN {X 0,Y 573.868,Z 496.78,A -85,B 0,C 180,E1 -2002.988,E2 -2002.988} C_VEL
LIN {X 0,Y 573.526,Z 500.357,A -85,B 0,C 180,E1 -2003.189,E2 -2003.189} C_VEL
LIN {X 0,Y 573.412,Z 511.674,A -85,B 0,C 180,E1 -2003.954,E2 -2003.954} C_VEL
LIN {X 0,Y 573.281,Z 521.815,A -85,B 0,C 180,E1 -2004.811,E2 -2004.811} C_VEL
LIN {X 0,Y 573.175,Z 529.608,A -85,B 0,C 180,E1 -2005.609,E2 -2005.609} C_VEL
LIN {X 0,Y 573.136,Z 536.665,A -85,B 0,C 180,E1 -2006.471,E2 -2006.471} C_VEL
LIN {X 0,Y 573.082,Z 542.87,A -85,B 0,C 180,E1 -2007.38,E2 -2007.38} C_VEL
LIN {X 0,Y 573.052,Z 547.826,A -85,B 0,C 180,E1 -2008.252,E2 -2008.252} C_VEL
LIN {X 0,Y 573.027,Z 552.965,A -85,B 0,C 180,E1 -2009.38,E2 -2009.38} C_VEL
LIN {X 0,Y 572.981,Z 555.907,A -85,B 0,C 180,E1 -2010.192,E2 -2010.192} C_VEL
LIN {X 0,Y 572.97,Z 558.259,A -85,B 0,C 180,E1 -2011.009,E2 -2011.009} C_VEL
LIN {X 0,Y 572.957,Z 560.588,A -85,B 0,C 180,E1 -2012.181,E2 -2012.181} C_VEL
LIN {X 0,Y 572.949,Z 561.843,A -85,B 0,C 180,E1 -2013.504,E2 -2013.504} C_VEL
LIN {X 0,Y 572.947,Z 561.781,A -85,B 0,C 180,E1 -2014.729,E2 -2014.729} C_VEL
LIN {X 0,Y 572.927,Z 560.332,A -85,B 0,C 180,E1 -2016.073,E2 -2016.073} C_VEL
LIN {X 0,Y 572.989,Z 557.27,A -85,B 0,C 180,E1 -2017.45,E2 -2017.45} C_VEL
LIN {X 0,Y 572.985,Z 552.917,A -85,B 0,C 180,E1 -2018.723,E2 -2018.723} C_VEL
LIN {X 0,Y 573.037,Z 547.797,A -85,B 0,C 180,E1 -2019.844,E2 -2019.844} C_VEL
LIN {X 0,Y 573.071,Z 541.024,A -85,B 0,C 180,E1 -2021.004,E2 -2021.004} C_VEL
LIN {X 0,Y 573.186,Z 532.215,A -85,B 0,C 180,E1 -2022.183,E2 -2022.183} C_VEL
LIN {X 0,Y 573.252,Z 524.029,A -85,B 0,C 180,E1 -2023.067,E2 -2023.067} C_VEL
LIN {X 0,Y 573.372,Z 514.983,A -85,B 0,C 180,E1 -2023.873,E2 -2023.873} C_VEL
LIN {X 0,Y 573.433,Z 506.44,A -85,B 0,C 180,E1 -2024.509,E2 -2024.509} C_VEL
LIN {X 0,Y 573.533,Z 496.646,A -85,B 0,C 180,E1 -2025.111,E2 -2025.111} C_VEL
LIN {X 0,Y 573.684,Z 486.035,A -85,B 0,C 180,E1 -2025.635,E2 -2025.635} C_VEL
LIN {X 0,Y 573.718,Z 479.671,A -85,B 0,C 180,E1 -2025.894,E2 -2025.894} C_VEL
LIN {X 0,Y 573.281,Z 477.076,A -85,B 0,C 180,E1 -2026.01,E2 -2026.01} C_VEL
LIN {X 0,Y 573.209,Z 477.083,A -85,B 0,C 180,E1 -2028.541,E2 -2028.541} C_VEL
LIN {X 0,Y 573.246,Z 477.08,A -85,B 0,C 180,E1 -2031.298,E2 -2031.298} C_VEL
LIN {X 0,Y 573.192,Z 477.089,A -85,B 0,C 180,E1 -2034.022,E2 -2034.022} C_VEL
LIN {X 0,Y 573.276,Z 477.075,A -85,B 0,C 180,E1 -2036.518,E2 -2036.518} C_VEL
LIN {X 0,Y 573.226,Z 477.081,A -85,B 0,C 180,E1 -2039.119,E2 -2039.119} C_VEL
LIN {X 0,Y 573.257,Z 477.077,A -85,B 0,C 180,E1 -2041.971,E2 -2041.971} C_VEL
LIN {X 0,Y 573.25,Z 477.081,A -85,B 0,C 180,E1 -2044.589,E2 -2044.589} C_VEL
LIN {X 0,Y 573.239,Z 477.081,A -85,B 0,C 180,E1 -2047.662,E2 -2047.662} C_VEL
LIN {X 0,Y 573.272,Z 477.077,A -85,B 0,C 180,E1 -2050.67,E2 -2050.67} C_VEL
LIN {X 0,Y 573.25,Z 477.08,A -85,B 0,C 180,E1 -2053.622,E2 -2053.622} C_VEL
LIN {X 0,Y 573.264,Z 477.076,A -85,B 0,C 180,E1 -2055.807,E2 -2055.807} C_VEL
LIN {X 0,Y 573.27,Z 477.075,A -85,B 0,C 180,E1 -2058.745,E2 -2058.745} C_VEL
LIN {X 0,Y 573.261,Z 477.076,A -85,B 0,C 180,E1 -2061.54,E2 -2061.54} C_VEL
LIN {X 0,Y 573.278,Z 477.074,A -85,B 0,C 180,E1 -2064.372,E2 -2064.372} C_VEL
LIN {X 0,Y 573.303,Z 477.073,A -85,B 0,C 180,E1 -2067.189,E2 -2067.189} C_VEL
LIN {X 0,Y 573.327,Z 477.071,A -85,B 0,C 180,E1 -2070,E2 -2070} C_VEL
LIN {X 0,Y 573.306,Z 477.075,A -85,B 0,C 180,E1 -2072.811,E2 -2072.811} C_VEL
LIN {X 0,Y 573.279,Z 477.077,A -85,B 0,C 180,E1 -2075.628,E2 -2075.628} C_VEL
LIN {X 0,Y 573.288,Z 477.074,A -85,B 0,C 180,E1 -2078.459,E2 -2078.459} C_VEL
LIN {X 0,Y 573.279,Z 477.075,A -85,B 0,C 180,E1 -2081.312,E2 -2081.312} C_VEL
LIN {X 0,Y 573.289,Z 477.074,A -85,B 0,C 180,E1 -2084.424,E2 -2084.424} C_VEL
LIN {X 0,Y 573.252,Z 477.077,A -85,B 0,C 180,E1 -2087.112,E2 -2087.112} C_VEL
LIN {X 0,Y 573.248,Z 477.077,A -85,B 0,C 180,E1 -2090.077,E2 -2090.077} C_VEL
LIN {X 0,Y 573.236,Z 477.084,A -85,B 0,C 180,E1 -2092.338,E2 -2092.338} C_VEL
LIN {X 0,Y 573.244,Z 477.082,A -85,B 0,C 180,E1 -2095.411,E2 -2095.411} C_VEL
LIN {X 0,Y 573.227,Z 477.083,A -85,B 0,C 180,E1 -2098.565,E2 -2098.565} C_VEL
LIN {X 0,Y 573.226,Z 477.083,A -85,B 0,C 180,E1 -2100.993,E2 -2100.993} C_VEL
LIN {X 0,Y 573.246,Z 477.078,A -85,B 0,C 180,E1 -2103.52,E2 -2103.52} C_VEL
LIN {X 0,Y 573.193,Z 477.086,A -85,B 0,C 180,E1 -2106.053,E2 -2106.053} C_VEL
LIN {X 0,Y 573.244,Z 477.083,A -85,B 0,C 180,E1 -2108.702,E2 -2108.702} C_VEL
LIN {X 0,Y 573.209,Z 477.087,A -85,B 0,C 180,E1 -2111.59,E2 -2111.59} C_VEL
LIN {X 0,Y 573.235,Z 477.08,A -85,B 0,C 180,E1 -2114.334,E2 -2114.334} C_VEL
LIN {X 0,Y 573.234,Z 477.081,A -85,B 0,C 180,E1 -2117.359,E2 -2117.359} C_VEL
LIN {X 0,Y 573.242,Z 477.08,A -85,B 0,C 180,E1 -2120.392,E2 -2120.392} C_VEL
LIN {X 0,Y 573.225,Z 477.081,A -85,B 0,C 180,E1 -2123.075,E2 -2123.075} C_VEL
LIN {X 0,Y 573.273,Z 477.075,A -85,B 0,C 180,E1 -2125.671,E2 -2125.671} C_VEL
LIN {X 0,Y 573.24,Z 477.084,A -85,B 0,C 180,E1 -2128.184,E2 -2128.184} C_VEL
LIN {X 0,Y 573.268,Z 477.076,A -85,B 0,C 180,E1 -2130.634,E2 -2130.634} C_VEL
LIN {X 0,Y 573.212,Z 477.084,A -85,B 0,C 180,E1 -2133.022,E2 -2133.022} C_VEL
LIN {X 0,Y 573.277,Z 477.076,A -85,B 0,C 180,E1 -2135.366,E2 -2135.366} C_VEL
LIN {X 0,Y 573.233,Z 477.082,A -85,B 0,C 180,E1 -2138.419,E2 -2138.419} C_VEL
LIN {X 0,Y 573.273,Z 477.075,A -85,B 0,C 180,E1 -2140.731,E2 -2140.731} C_VEL
LIN {X 0,Y 573.247,Z 477.078,A -85,B 0,C 180,E1 -2143.621,E2 -2143.621} C_VEL
LIN {X 0,Y 573.26,Z 477.078,A -85,B 0,C 180,E1 -2145.806,E2 -2145.806} C_VEL
LIN {X 0,Y 573.267,Z 477.077,A -85,B 0,C 180,E1 -2148.745,E2 -2148.745} C_VEL
LIN {X 0,Y 573.254,Z 477.077,A -85,B 0,C 180,E1 -2151.54,E2 -2151.54} C_VEL
LIN {X 0,Y 573.285,Z 477.073,A -85,B 0,C 180,E1 -2154.372,E2 -2154.372} C_VEL
LIN {X 0,Y 573.312,Z 477.073,A -85,B 0,C 180,E1 -2157.892,E2 -2157.892} C_VEL
LIN {X 0,Y 573.33,Z 477.069,A -85,B 0,C 180,E1 -2160.702,E2 -2160.702} C_VEL
LIN {X 0,Y 573.299,Z 477.074,A -85,B 0,C 180,E1 -2162.81,E2 -2162.81} C_VEL
LIN {X 0,Y 573.282,Z 477.078,A -85,B 0,C 180,E1 -2165.628,E2 -2165.628} C_VEL
LIN {X 0,Y 573.284,Z 477.077,A -85,B 0,C 180,E1 -2168.459,E2 -2168.459} C_VEL
LIN {X 0,Y 573.275,Z 477.077,A -85,B 0,C 180,E1 -2171.312,E2 -2171.312} C_VEL
LIN {X 0,Y 573.263,Z 477.077,A -85,B 0,C 180,E1 -2174.193,E2 -2174.193} C_VEL
LIN {X 0,Y 573.252,Z 477.078,A -85,B 0,C 180,E1 -2177.112,E2 -2177.112} C_VEL
LIN {X 0,Y 573.246,Z 477.078,A -85,B 0,C 180,E1 -2180.077,E2 -2180.077} C_VEL
LIN {X 0,Y 573.221,Z 477.083,A -85,B 0,C 180,E1 -2182.338,E2 -2182.338} C_VEL
LIN {X 0,Y 573.27,Z 477.079,A -85,B 0,C 180,E1 -2184.878,E2 -2184.878} C_VEL
LIN {X 0,Y 573.232,Z 477.082,A -85,B 0,C 180,E1 -2187.768,E2 -2187.768} C_VEL
LIN {X 0,Y 573.247,Z 477.078,A -85,B 0,C 180,E1 -2190.176,E2 -2190.176} C_VEL
LIN {X 0,Y 573.255,Z 477.081,A -85,B 0,C 180,E1 -2192.645,E2 -2192.645} C_VEL
LIN {X 0,Y 573.205,Z 477.085,A -85,B 0,C 180,E1 -2195.188,E2 -2195.188} C_VEL
LIN {X 0,Y 573.236,Z 477.078,A -85,B 0,C 180,E1 -2197.808,E2 -2197.808} C_VEL
LIN {X 0,Y 573.247,Z 477.078,A -85,B 0,C 180,E1 -2200.525,E2 -2200.525} C_VEL
LIN {X 0,Y 573.239,Z 477.08,A -85,B 0,C 180,E1 -2203.359,E2 -2203.359} C_VEL
LIN {X 0,Y 573.211,Z 477.083,A -85,B 0,C 180,E1 -2206.335,E2 -2206.335} C_VEL
LIN {X 0,Y 573.242,Z 477.078,A -85,B 0,C 180,E1 -2208.544,E2 -2208.544} C_VEL
LIN {X 0,Y 573.235,Z 477.08,A -85,B 0,C 180,E1 -2211.298,E2 -2211.298} C_VEL
LIN {X 0,Y 573.256,Z 477.283,A -85,B 0,C 180,E1 -2213.133,E2 -2213.133} C_VEL
LIN {X 0,Y 574.162,Z 482.24,A -85,B 0,C 180,E1 -2214.234,E2 -2214.234} C_VEL
LIN {X 0,Y 574.057,Z 495.574,A -85,B 0,C 180,E1 -2216.989,E2 -2216.989} C_VEL
LIN {X 0,Y 574.085,Z 510.171,A -85,B 0,C 180,E1 -2219.872,E2 -2219.872} C_VEL
LIN {X 0,Y 573.973,Z 524.755,A -85,B 0,C 180,E1 -2222.667,E2 -2222.667} C_VEL
LIN {X 0,Y 573.849,Z 538.45,A -85,B 0,C 180,E1 -2225.392,E2 -2225.392} C_VEL
LIN {X 0,Y 573.62,Z 552.145,A -85,B 0,C 180,E1 -2228.057,E2 -2228.057} C_VEL
LIN {X 0,Y 573.481,Z 565.84,A -85,B 0,C 180,E1 -2230.678,E2 -2230.678} C_VEL
LIN {X 0,Y 573.362,Z 579.687,A -85,B 0,C 180,E1 -2233.287,E2 -2233.287} C_VEL
LIN {X 0,Y 573.243,Z 595.187,A -85,B 0,C 180,E1 -2236.168,E2 -2236.168} C_VEL
LIN {X 0,Y 573.197,Z 602.157,A -85,B 0,C 180,E1 -2237.452,E2 -2237.452} C_VEL
LIN {X 0,Y 573.864,Z 607.947,A -85,B 0,C 180,E1 -2237.557,E2 -2237.557} C_VEL
LIN {X 0,Y 573.807,Z 621.22,A -85,B 0,C 180,E1 -2237.87,E2 -2237.87} C_VEL
LIN {X 0,Y 573.702,Z 633.373,A -85,B 0,C 180,E1 -2238.294,E2 -2238.294} C_VEL
LIN {X 0,Y 573.574,Z 645.719,A -85,B 0,C 180,E1 -2238.878,E2 -2238.878} C_VEL
LIN {X 0,Y 573.433,Z 657.203,A -85,B 0,C 180,E1 -2239.585,E2 -2239.585} C_VEL
LIN {X 0,Y 573.334,Z 667.599,A -85,B 0,C 180,E1 -2240.386,E2 -2240.386} C_VEL
LIN {X 0,Y 573.241,Z 676.113,A -85,B 0,C 180,E1 -2241.185,E2 -2241.185} C_VEL
LIN {X 0,Y 573.161,Z 683.961,A -85,B 0,C 180,E1 -2242.071,E2 -2242.071} C_VEL
LIN {X 0,Y 573.072,Z 691.954,A -85,B 0,C 180,E1 -2243.185,E2 -2243.185} C_VEL
LIN {X 0,Y 573.07,Z 698.68,A -85,B 0,C 180,E1 -2244.37,E2 -2244.37} C_VEL
LIN {X 0,Y 573.028,Z 703.372,A -85,B 0,C 180,E1 -2245.428,E2 -2245.428} C_VEL
LIN {X 0,Y 573.022,Z 706.957,A -85,B 0,C 180,E1 -2246.484,E2 -2246.484} C_VEL
LIN {X 0,Y 572.959,Z 708.809,A -85,B 0,C 180,E1 -2247.188,E2 -2247.188} C_VEL
LIN {X 0,Y 572.939,Z 710.199,A -85,B 0,C 180,E1 -2247.891,E2 -2247.891} C_VEL
LIN {X 0,Y 572.94,Z 711.785,A -85,B 0,C 180,E1 -2249.297,E2 -2249.297} C_VEL
LIN {X 0,Y 572.938,Z 712,A -85,B 0,C 180,E1 -2250,E2 -2250} C_VEL
LIN {X 0,Y 572.946,Z 711.186,A -85,B 0,C 180,E1 -2251.406,E2 -2251.406} C_VEL
LIN {X 0,Y 572.939,Z 710.2,A -85,B 0,C 180,E1 -2252.109,E2 -2252.109} C_VEL
LIN {X 0,Y 572.959,Z 708.81,A -85,B 0,C 180,E1 -2252.812,E2 -2252.812} C_VEL
LIN {X 0,Y 573.015,Z 705.896,A -85,B 0,C 180,E1 -2253.868,E2 -2253.868} C_VEL
LIN {X 0,Y 572.963,Z 701.949,A -85,B 0,C 180,E1 -2254.926,E2 -2254.926} C_VEL
LIN {X 0,Y 573.064,Z 695.876,A -85,B 0,C 180,E1 -2256.16,E2 -2256.16} C_VEL
LIN {X 0,Y 573.119,Z 689.236,A -85,B 0,C 180,E1 -2257.221,E2 -2257.221} C_VEL
LIN {X 0,Y 573.201,Z 680.989,A -85,B 0,C 180,E1 -2258.283,E2 -2258.283} C_VEL
LIN {X 0,Y 573.287,Z 672.536,A -85,B 0,C 180,E1 -2259.17,E2 -2259.17} C_VEL
LIN {X 0,Y 573.43,Z 662.094,A -85,B 0,C 180,E1 -2260.058,E2 -2260.058} C_VEL
LIN {X 0,Y 573.549,Z 650.427,A -85,B 0,C 180,E1 -2260.853,E2 -2260.853} C_VEL
LIN {X 0,Y 573.641,Z 638.878,A -85,B 0,C 180,E1 -2261.466,E2 -2261.466} C_VEL
LIN {X 0,Y 573.732,Z 626.169,A -85,B 0,C 180,E1 -2261.975,E2 -2261.975} C_VEL
LIN {X 0,Y 573.852,Z 613.513,A -85,B 0,C 180,E1 -2262.331,E2 -2262.331} C_VEL
LIN {X 0,Y 573.675,Z 605.097,A -85,B 0,C 180,E1 -2262.492,E2 -2262.492} C_VEL
LIN {X 0,Y 573.203,Z 602.033,A -85,B 0,C 180,E1 -2262.57,E2 -2262.57} C_VEL
LIN {X 0,Y 573.31,Z 585.404,A -85,B 0,C 180,E1 -2265.646,E2 -2265.646} C_VEL
LIN {X 0,Y 573.459,Z 571.709,A -85,B 0,C 180,E1 -2268.211,E2 -2268.211} C_VEL
LIN {X 0,Y 573.597,Z 555.076,A -85,B 0,C 180,E1 -2271.378,E2 -2271.378} C_VEL
LIN {X 0,Y 573.794,Z 540.406,A -85,B 0,C 180,E1 -2274.225,E2 -2274.225} C_VEL
LIN {X 0,Y 573.949,Z 526.711,A -85,B 0,C 180,E1 -2276.941,E2 -2276.941} C_VEL
LIN {X 0,Y 573.992,Z 517.292,A -85,B 0,C 180,E1 -2278.724,E2 -2278.724} C_VEL
LIN {X 0,Y 573.909,Z 503.259,A -85,B 0,C 180,E1 -2281.362,E2 -2281.362} C_VEL
LIN {X 0,Y 573.889,Z 488.074,A -85,B 0,C 180,E1 -2284.287,E2 -2284.287} C_VEL
LIN {X 0,Y 573.837,Z 480.59,A -85,B 0,C 180,E1 -2285.79,E2 -2285.79} C_VEL
LIN {X 0,Y 573.222,Z 477.085,A -85,B 0,C 180,E1 -2286.569,E2 -2286.569} C_VEL
LIN {X 0,Y 573.245,Z 477.08,A -85,B 0,C 180,E1 -2289.432,E2 -2289.432} C_VEL
LIN {X 0,Y 573.243,Z 477.084,A -85,B 0,C 180,E1 -2292.401,E2 -2292.401} C_VEL
LIN {X 0,Y 573.23,Z 477.083,A -85,B 0,C 180,E1 -2295.325,E2 -2295.325} C_VEL
LIN {X 0,Y 573.243,Z 477.083,A -85,B 0,C 180,E1 -2297.6,E2 -2297.6} C_VEL
LIN {X 0,Y 573.246,Z 477.08,A -85,B 0,C 180,E1 -2300.569,E2 -2300.569} C_VEL
LIN {X 0,Y 573.235,Z 477.081,A -85,B 0,C 180,E1 -2303.076,E2 -2303.076} C_VEL
LIN {X 0,Y 573.263,Z 477.078,A -85,B 0,C 180,E1 -2305.671,E2 -2305.671} C_VEL
LIN {X 0,Y 573.245,Z 477.079,A -85,B 0,C 180,E1 -2308.185,E2 -2308.185} C_VEL
LIN {X 0,Y 573.267,Z 477.076,A -85,B 0,C 180,E1 -2310.634,E2 -2310.634} C_VEL
LIN {X 0,Y 573.238,Z 477.083,A -85,B 0,C 180,E1 -2313.508,E2 -2313.508} C_VEL
LIN {X 0,Y 573.231,Z 477.084,A -85,B 0,C 180,E1 -2316.135,E2 -2316.135} C_VEL
LIN {X 0,Y 573.252,Z 477.078,A -85,B 0,C 180,E1 -2319.174,E2 -2319.174} C_VEL
LIN {X 0,Y 573.223,Z 477.083,A -85,B 0,C 180,E1 -2321.411,E2 -2321.411} C_VEL
LIN {X 0,Y 573.25,Z 477.082,A -85,B 0,C 180,E1 -2323.622,E2 -2323.622} C_VEL
LIN {X 0,Y 573.23,Z 477.082,A -85,B 0,C 180,E1 -2326.529,E2 -2326.529} C_VEL
LIN {X 0,Y 573.268,Z 477.078,A -85,B 0,C 180,E1 -2328.745,E2 -2328.745} C_VEL
LIN {X 0,Y 573.287,Z 477.074,A -85,B 0,C 180,E1 -2331.541,E2 -2331.541} C_VEL
LIN {X 0,Y 573.298,Z 477.074,A -85,B 0,C 180,E1 -2334.372,E2 -2334.372} C_VEL
LIN {X 0,Y 573.316,Z 477.071,A -85,B 0,C 180,E1 -2337.893,E2 -2337.893} C_VEL
LIN {X 0,Y 573.334,Z 477.07,A -85,B 0,C 180,E1 -2340.703,E2 -2340.703} C_VEL
LIN {X 0,Y 573.301,Z 477.073,A -85,B 0,C 180,E1 -2342.811,E2 -2342.811} C_VEL
LIN {X 0,Y 573.281,Z 477.076,A -85,B 0,C 180,E1 -2345.628,E2 -2345.628} C_VEL
LIN {X 0,Y 573.287,Z 477.078,A -85,B 0,C 180,E1 -2348.46,E2 -2348.46} C_VEL
LIN {X 0,Y 573.278,Z 477.076,A -85,B 0,C 180,E1 -2351.312,E2 -2351.312} C_VEL
LIN {X 0,Y 573.288,Z 477.076,A -85,B 0,C 180,E1 -2354.425,E2 -2354.425} C_VEL
LIN {X 0,Y 573.264,Z 477.082,A -85,B 0,C 180,E1 -2357.112,E2 -2357.112} C_VEL
LIN {X 0,Y 573.246,Z 477.081,A -85,B 0,C 180,E1 -2360.077,E2 -2360.077} C_VEL
LIN {X 0,Y 573.264,Z 477.21,A -85,B 0,C 180,E1 -2362.1,E2 -2362.1} C_VEL
LIN {X 0,Y 573.72,Z 480.451,A -85,B 0,C 180,E1 -2362.223,E2 -2362.223} C_VEL
LIN {X 0,Y 573.593,Z 493.358,A -85,B 0,C 180,E1 -2362.799,E2 -2362.799} C_VEL
LIN {X 0,Y 573.526,Z 500.357,A -85,B 0,C 180,E1 -2363.189,E2 -2363.189} C_VEL
LIN {X 0,Y 572.811,Z 505.408,A -85,B 0,C 180,E1 -2363.487,E2 -2363.487} C_VEL
LIN {X 0,Y 569.887,Z 513.306,A -85,B 0,C 180,E1 -2364.013,E2 -2364.013} C_VEL
LIN {X 0,Y 566.937,Z 520.773,A -85,B 0,C 180,E1 -2364.607,E2 -2364.607} C_VEL
LIN {X 0,Y 566.187,Z 525.037,A -85,B 0,C 180,E1 -2365.01,E2 -2365.01} C_VEL
LIN {X 0,Y 566.08,Z 534.992,A -85,B 0,C 180,E1 -2366.151,E2 -2366.151} C_VEL
LIN {X 0,Y 566.007,Z 541.99,A -85,B 0,C 180,E1 -2367.153,E2 -2367.153} C_VEL
LIN {X 0,Y 565.966,Z 547.704,A -85,B 0,C 180,E1 -2368.156,E2 -2368.156} C_VEL
LIN {X 0,Y 565.94,Z 552.848,A -85,B 0,C 180,E1 -2369.293,E2 -2369.293} C_VEL
LIN {X 0,Y 565.901,Z 556.064,A -85,B 0,C 180,E1 -2370.197,E2 -2370.197} C_VEL
LIN {X 0,Y 565.845,Z 559.296,A -85,B 0,C 180,E1 -2371.444,E2 -2371.444} C_VEL
LIN {X 0,Y 565.849,Z 560.86,A -85,B 0,C 180,E1 -2372.373,E2 -2372.373} C_VEL
LIN {X 0,Y 565.855,Z 561.912,A -85,B 0,C 180,E1 -2373.679,E2 -2373.679} C_VEL
LIN {X 0,Y 565.84,Z 561.666,A -85,B 0,C 180,E1 -2374.939,E2 -2374.939} C_VEL
LIN {X 0,Y 565.827,Z 560.235,A -85,B 0,C 180,E1 -2376.162,E2 -2376.162} C_VEL
LIN {X 0,Y 565.915,Z 557.295,A -85,B 0,C 180,E1 -2377.483,E2 -2377.483} C_VEL
LIN {X 0,Y 565.893,Z 553.964,A -85,B 0,C 180,E1 -2378.517,E2 -2378.517} C_VEL
LIN {X 0,Y 565.968,Z 549.095,A -85,B 0,C 180,E1 -2379.655,E2 -2379.655} C_VEL
LIN {X 0,Y 565.994,Z 544.729,A -85,B 0,C 180,E1 -2380.487,E2 -2380.487} C_VEL
LIN {X 0,Y 566.03,Z 538.218,A -85,B 0,C 180,E1 -2381.501,E2 -2381.501} C_VEL
